LIN {X 0,Y 374.642,Z 535.942,A -85,B 0,C 180,E1 -12888.125,E2 -12888.125} C_VEL
LIN {X 0,Y 374.323,Z 532.294,A -85,B 0,C 180,E1 -12888.371,E2 -12888.371} C_VEL
LIN {X 0,Y 371.906,Z 526.656,A -85,B 0,C 180,E1 -12888.815,E2 -12888.815} C_VEL
LIN {X 0,Y 369.429,Z 520.933,A -85,B 0,C 180,E1 -12889.223,E2 -12889.223} C_VEL
LIN {X 0,Y 368.959,Z 517.153,A -85,B 0,C 180,E1 -12889.399,E2 -12889.399} C_VEL
LIN {X 0,Y 369.367,Z 505.054,A -85,B 0,C 180,E1 -12889.739,E2 -12889.739} C_VEL
LIN {X 0,Y 370.451,Z 429.303,A -85,B 0,C 180,E1 -12891.218,E2 -12891.218} C_VEL
LIN {X 0,Y 365.654,Z 406.161,A -85,B 0,C 180,E1 -12891.992,E2 -12891.992} C_VEL
LIN {X 0,Y 364.747,Z 403.294,A -85,B 0,C 180,E1 -12892.123,E2 -12892.123} C_VEL
LIN {X 0,Y 362.511,Z 391.552,A -85,B 0,C 180,E1 -12895.554,E2 -12895.554} C_VEL
LIN {X 0,Y 361.948,Z 388.902,A -85,B 0,C 180,E1 -12896.37,E2 -12896.37} C_VEL
LIN {X 0,Y 361.916,Z 388.903,A -85,B 0,C 180,E1 -12899.09,E2 -12899.09} C_VEL
LIN {X 0,Y 361.852,Z 388.912,A -85,B 0,C 180,E1 -12902.945,E2 -12902.945} C_VEL
LIN {X 0,Y 361.871,Z 388.905,A -85,B 0,C 180,E1 -12905.637,E2 -12905.637} C_VEL
LIN {X 0,Y 361.873,Z 388.908,A -85,B 0,C 180,E1 -12909.027,E2 -12909.027} C_VEL
LIN {X 0,Y 361.839,Z 388.913,A -85,B 0,C 180,E1 -12912.829,E2 -12912.829} C_VEL
LIN {X 0,Y 361.825,Z 388.912,A -85,B 0,C 180,E1 -12915.946,E2 -12915.946} C_VEL
LIN {X 0,Y 361.859,Z 388.907,A -85,B 0,C 180,E1 -12919.241,E2 -12919.241} C_VEL
LIN {X 0,Y 361.875,Z 388.908,A -85,B 0,C 180,E1 -12922.776,E2 -12922.776} C_VEL
LIN {X 0,Y 361.858,Z 388.907,A -85,B 0,C 180,E1 -12925.72,E2 -12925.72} C_VEL
LIN {X 0,Y 361.88,Z 388.905,A -85,B 0,C 180,E1 -12929.672,E2 -12929.672} C_VEL
LIN {X 0,Y 361.959,Z 388.895,A -85,B 0,C 180,E1 -12933.475,E2 -12933.475} C_VEL
LIN {X 0,Y 361.897,Z 388.902,A -85,B 0,C 180,E1 -12937.145,E2 -12937.145} C_VEL
LIN {X 0,Y 361.933,Z 388.898,A -85,B 0,C 180,E1 -12940.725,E2 -12940.725} C_VEL
LIN {X 0,Y 361.951,Z 388.9,A -85,B 0,C 180,E1 -12944.226,E2 -12944.226} C_VEL
LIN {X 0,Y 362.003,Z 388.89,A -85,B 0,C 180,E1 -12946.528,E2 -12946.528} C_VEL
LIN {X 0,Y 362.036,Z 388.891,A -85,B 0,C 180,E1 -12949.938,E2 -12949.938} C_VEL
LIN {X 0,Y 362.156,Z 388.873,A -85,B 0,C 180,E1 -12952.193,E2 -12952.193} C_VEL
LIN {X 0,Y 362.123,Z 388.875,A -85,B 0,C 180,E1 -12954.431,E2 -12954.431} C_VEL
LIN {X 0,Y 362.286,Z 388.859,A -85,B 0,C 180,E1 -12957.776,E2 -12957.776} C_VEL
LIN {X 0,Y 362.431,Z 388.84,A -85,B 0,C 180,E1 -12960,E2 -12960} C_VEL
LIN {X 0,Y 362.286,Z 388.856,A -85,B 0,C 180,E1 -12962.223,E2 -12962.223} C_VEL
LIN {X 0,Y 362.157,Z 388.87,A -85,B 0,C 180,E1 -12966.686,E2 -12966.686} C_VEL
LIN {X 0,Y 362.037,Z 388.887,A -85,B 0,C 180,E1 -12970.062,E2 -12970.062} C_VEL
LIN {X 0,Y 362.003,Z 388.892,A -85,B 0,C 180,E1 -12973.899,E2 -12973.899} C_VEL
LIN {X 0,Y 361.971,Z 388.895,A -85,B 0,C 180,E1 -12977.938,E2 -12977.938} C_VEL
LIN {X 0,Y 361.897,Z 388.906,A -85,B 0,C 180,E1 -12981.653,E2 -12981.653} C_VEL
LIN {X 0,Y 361.932,Z 388.903,A -85,B 0,C 180,E1 -12985.29,E2 -12985.29} C_VEL
LIN {X 0,Y 361.912,Z 388.902,A -85,B 0,C 180,E1 -12987.779,E2 -12987.779} C_VEL
LIN {X 0,Y 361.841,Z 388.912,A -85,B 0,C 180,E1 -12991.629,E2 -12991.629} C_VEL
LIN {X 0,Y 361.877,Z 388.91,A -85,B 0,C 180,E1 -12995.345,E2 -12995.345} C_VEL
LIN {X 0,Y 361.872,Z 388.91,A -85,B 0,C 180,E1 -12999.026,E2 -12999.026} C_VEL
LIN {X 0,Y 361.84,Z 388.912,A -85,B 0,C 180,E1 -13002.828,E2 -13002.828} C_VEL
LIN {X 0,Y 361.831,Z 388.91,A -85,B 0,C 180,E1 -13005.945,E2 -13005.945} C_VEL
LIN {X 0,Y 361.839,Z 388.913,A -85,B 0,C 180,E1 -13009.244,E2 -13009.244} C_VEL
LIN {X 0,Y 361.867,Z 388.91,A -85,B 0,C 180,E1 -13012.777,E2 -13012.777} C_VEL
LIN {X 0,Y 361.857,Z 388.907,A -85,B 0,C 180,E1 -13015.719,E2 -13015.719} C_VEL
LIN {X 0,Y 361.882,Z 388.909,A -85,B 0,C 180,E1 -13019.672,E2 -13019.672} C_VEL
LIN {X 0,Y 361.935,Z 389.076,A -85,B 0,C 180,E1 -13020.317,E2 -13020.317} C_VEL
LIN {X 0,Y 364.172,Z 399.647,A -85,B 0,C 180,E1 -13023.187,E2 -13023.187} C_VEL
LIN {X 0,Y 365.709,Z 407.696,A -85,B 0,C 180,E1 -13025.293,E2 -13025.293} C_VEL
LIN {X 0,Y 364.82,Z 417.446,A -85,B 0,C 180,E1 -13027.621,E2 -13027.621} C_VEL
LIN {X 0,Y 364.736,Z 418.695,A -85,B 0,C 180,E1 -13027.921,E2 -13027.921} C_VEL
LIN {X 0,Y 369.876,Z 448.618,A -85,B 0,C 180,E1 -13028.855,E2 -13028.855} C_VEL
LIN {X 0,Y 370.27,Z 453.848,A -85,B 0,C 180,E1 -13028.985,E2 -13028.985} C_VEL
LIN {X 0,Y 369.021,Z 526.846,A -85,B 0,C 180,E1 -13030.423,E2 -13030.423} C_VEL
LIN {X 0,Y 368.4,Z 539.299,A -85,B 0,C 180,E1 -13030.859,E2 -13030.859} C_VEL
LIN {X 0,Y 367.479,Z 552.192,A -85,B 0,C 180,E1 -13031.533,E2 -13031.533} C_VEL
LIN {X 0,Y 366.459,Z 564.435,A -85,B 0,C 180,E1 -13032.419,E2 -13032.419} C_VEL
LIN {X 0,Y 365.313,Z 576.016,A -85,B 0,C 180,E1 -13033.515,E2 -13033.515} C_VEL
LIN {X 0,Y 364.277,Z 586.157,A -85,B 0,C 180,E1 -13034.721,E2 -13034.721} C_VEL
LIN {X 0,Y 363.413,Z 594.976,A -85,B 0,C 180,E1 -13036.011,E2 -13036.011} C_VEL
LIN {X 0,Y 362.534,Z 602.845,A -85,B 0,C 180,E1 -13037.403,E2 -13037.403} C_VEL
LIN {X 0,Y 361.629,Z 610.529,A -85,B 0,C 180,E1 -13039.077,E2 -13039.077} C_VEL
LIN {X 0,Y 360.954,Z 617.618,A -85,B 0,C 180,E1 -13041.039,E2 -13041.039} C_VEL
LIN {X 0,Y 360.601,Z 622.335,A -85,B 0,C 180,E1 -13042.722,E2 -13042.722} C_VEL
LIN {X 0,Y 360.383,Z 625.939,A -85,B 0,C 180,E1 -13044.404,E2 -13044.404} C_VEL
LIN {X 0,Y 360.346,Z 627.799,A -85,B 0,C 180,E1 -13045.525,E2 -13045.525} C_VEL
LIN {X 0,Y 360.29,Z 629.193,A -85,B 0,C 180,E1 -13046.645,E2 -13046.645} C_VEL
LIN {X 0,Y 360.289,Z 630.795,A -85,B 0,C 180,E1 -13048.882,E2 -13048.882} C_VEL
LIN {X 0,Y 360.311,Z 631.01,A -85,B 0,C 180,E1 -13050,E2 -13050} C_VEL
LIN {X 0,Y 360.289,Z 630.792,A -85,B 0,C 180,E1 -13051.118,E2 -13051.118} C_VEL
LIN {X 0,Y 360.29,Z 629.185,A -85,B 0,C 180,E1 -13053.355,E2 -13053.355} C_VEL
LIN {X 0,Y 360.346,Z 627.787,A -85,B 0,C 180,E1 -13054.474,E2 -13054.474} C_VEL
LIN {X 0,Y 360.382,Z 625.21,A -85,B 0,C 180,E1 -13055.968,E2 -13055.968} C_VEL
LIN {X 0,Y 360.697,Z 620.874,A -85,B 0,C 180,E1 -13057.839,E2 -13057.839} C_VEL
LIN {X 0,Y 361.197,Z 614.761,A -85,B 0,C 180,E1 -13059.802,E2 -13059.802} C_VEL
LIN {X 0,Y 361.868,Z 608.085,A -85,B 0,C 180,E1 -13061.482,E2 -13061.482} C_VEL
LIN {X 0,Y 362.864,Z 599.806,A -85,B 0,C 180,E1 -13063.154,E2 -13063.154} C_VEL
LIN {X 0,Y 363.732,Z 591.315,A -85,B 0,C 180,E1 -13064.548,E2 -13064.548} C_VEL
LIN {X 0,Y 364.806,Z 580.824,A -85,B 0,C 180,E1 -13065.934,E2 -13065.934} C_VEL
LIN {X 0,Y 365.981,Z 569.017,A -85,B 0,C 180,E1 -13067.172,E2 -13067.172} C_VEL
LIN {X 0,Y 367.024,Z 557.134,A -85,B 0,C 180,E1 -13068.129,E2 -13068.129} C_VEL
LIN {X 0,Y 368.02,Z 544.771,A -85,B 0,C 180,E1 -13068.872,E2 -13068.872} C_VEL
LIN {X 0,Y 368.758,Z 532.06,A -85,B 0,C 180,E1 -13069.41,E2 -13069.41} C_VEL
LIN {X 0,Y 369.217,Z 518.696,A -85,B 0,C 180,E1 -13069.747,E2 -13069.747} C_VEL
LIN {X 0,Y 370.129,Z 450.447,A -85,B 0,C 180,E1 -13071.079,E2 -13071.079} C_VEL
LIN {X 0,Y 365.387,Z 422.391,A -85,B 0,C 180,E1 -13071.944,E2 -13071.944} C_VEL
LIN {X 0,Y 364.722,Z 418.661,A -85,B 0,C 180,E1 -13072.071,E2 -13072.071} C_VEL
LIN {X 0,Y 365.716,Z 408.872,A -85,B 0,C 180,E1 -13074.404,E2 -13074.404} C_VEL
LIN {X 0,Y 364.791,Z 402.605,A -85,B 0,C 180,E1 -13076.014,E2 -13076.014} C_VEL
LIN {X 0,Y 362.303,Z 390.756,A -85,B 0,C 180,E1 -13079.2,E2 -13079.2} C_VEL
LIN {X 0,Y 361.893,Z 388.903,A -85,B 0,C 180,E1 -13079.764,E2 -13079.764} C_VEL
LIN {X 0,Y 361.86,Z 388.91,A -85,B 0,C 180,E1 -13083.369,E2 -13083.369} C_VEL
LIN {X 0,Y 361.869,Z 388.912,A -85,B 0,C 180,E1 -13087.018,E2 -13087.018} C_VEL
LIN {X 0,Y 361.857,Z 388.907,A -85,B 0,C 180,E1 -13089.861,E2 -13089.861} C_VEL
LIN {X 0,Y 361.837,Z 388.915,A -85,B 0,C 180,E1 -13092.829,E2 -13092.829} C_VEL
LIN {X 0,Y 361.83,Z 388.91,A -85,B 0,C 180,E1 -13095.945,E2 -13095.945} C_VEL
LIN {X 0,Y 361.838,Z 388.912,A -85,B 0,C 180,E1 -13099.244,E2 -13099.244} C_VEL
LIN {X 0,Y 361.865,Z 388.912,A -85,B 0,C 180,E1 -13102.777,E2 -13102.777} C_VEL
LIN {X 0,Y 361.856,Z 388.907,A -85,B 0,C 180,E1 -13105.72,E2 -13105.72} C_VEL
LIN {X 0,Y 361.874,Z 388.905,A -85,B 0,C 180,E1 -13109.672,E2 -13109.672} C_VEL
LIN {X 0,Y 361.955,Z 388.895,A -85,B 0,C 180,E1 -13113.475,E2 -13113.475} C_VEL
LIN {X 0,Y 361.894,Z 388.904,A -85,B 0,C 180,E1 -13117.145,E2 -13117.145} C_VEL
LIN {X 0,Y 361.909,Z 388.905,A -85,B 0,C 180,E1 -13120.723,E2 -13120.723} C_VEL
LIN {X 0,Y 361.935,Z 388.898,A -85,B 0,C 180,E1 -13123.066,E2 -13123.066} C_VEL
LIN {X 0,Y 362.003,Z 388.894,A -85,B 0,C 180,E1 -13126.528,E2 -13126.528} C_VEL
LIN {X 0,Y 362.035,Z 388.887,A -85,B 0,C 180,E1 -13129.938,E2 -13129.938} C_VEL
LIN {X 0,Y 362.153,Z 388.87,A -85,B 0,C 180,E1 -13133.314,E2 -13133.314} C_VEL
LIN {X 0,Y 362.283,Z 388.856,A -85,B 0,C 180,E1 -13137.777,E2 -13137.777} C_VEL
LIN {X 0,Y 362.429,Z 388.84,A -85,B 0,C 180,E1 -13140,E2 -13140} C_VEL
LIN {X 0,Y 362.286,Z 388.86,A -85,B 0,C 180,E1 -13142.224,E2 -13142.224} C_VEL
LIN {X 0,Y 362.175,Z 388.868,A -85,B 0,C 180,E1 -13146.686,E2 -13146.686} C_VEL
LIN {X 0,Y 362.076,Z 388.88,A -85,B 0,C 180,E1 -13148.933,E2 -13148.933} C_VEL
LIN {X 0,Y 361.963,Z 388.897,A -85,B 0,C 180,E1 -13152.332,E2 -13152.332} C_VEL
LIN {X 0,Y 361.964,Z 388.894,A -85,B 0,C 180,E1 -13154.62,E2 -13154.62} C_VEL
LIN {X 0,Y 361.963,Z 388.898,A -85,B 0,C 180,E1 -13158.099,E2 -13158.099} C_VEL
LIN {X 0,Y 361.901,Z 388.905,A -85,B 0,C 180,E1 -13161.652,E2 -13161.652} C_VEL
LIN {X 0,Y 361.93,Z 388.899,A -85,B 0,C 180,E1 -13165.29,E2 -13165.29} C_VEL
LIN {X 0,Y 361.925,Z 388.905,A -85,B 0,C 180,E1 -13167.778,E2 -13167.778} C_VEL
LIN {X 0,Y 361.849,Z 388.91,A -85,B 0,C 180,E1 -13171.285,E2 -13171.285} C_VEL
LIN {X 0,Y 361.857,Z 388.908,A -85,B 0,C 180,E1 -13174.28,E2 -13174.28} C_VEL
LIN {X 0,Y 361.873,Z 388.907,A -85,B 0,C 180,E1 -13177.225,E2 -13177.225} C_VEL
LIN {X 0,Y 361.857,Z 388.907,A -85,B 0,C 180,E1 -13180.759,E2 -13180.759} C_VEL
LIN {X 0,Y 361.82,Z 388.912,A -85,B 0,C 180,E1 -13184.368,E2 -13184.368} C_VEL
LIN {X 0,Y 361.838,Z 388.915,A -85,B 0,C 180,E1 -13187.568,E2 -13187.568} C_VEL
LIN {X 0,Y 361.872,Z 388.907,A -85,B 0,C 180,E1 -13190.973,E2 -13190.973} C_VEL
LIN {X 0,Y 361.877,Z 388.905,A -85,B 0,C 180,E1 -13194.655,E2 -13194.655} C_VEL
LIN {X 0,Y 361.839,Z 388.909,A -85,B 0,C 180,E1 -13198.371,E2 -13198.371} C_VEL
LIN {X 0,Y 361.902,Z 388.905,A -85,B 0,C 180,E1 -13200.955,E2 -13200.955} C_VEL
LIN {X 0,Y 361.983,Z 389.022,A -85,B 0,C 180,E1 -13203.788,E2 -13203.788} C_VEL
LIN {X 0,Y 364.099,Z 399.857,A -85,B 0,C 180,E1 -13206.991,E2 -13206.991} C_VEL
LIN {X 0,Y 364.792,Z 403.485,A -85,B 0,C 180,E1 -13208.002,E2 -13208.002} C_VEL
LIN {X 0,Y 367.169,Z 412.809,A -85,B 0,C 180,E1 -13208.346,E2 -13208.346} C_VEL
LIN {X 0,Y 370.497,Z 429.487,A -85,B 0,C 180,E1 -13208.892,E2 -13208.892} C_VEL
LIN {X 0,Y 369.404,Z 500.103,A -85,B 0,C 180,E1 -13210.263,E2 -13210.263} C_VEL
LIN {X 0,Y 369.09,Z 514.346,A -85,B 0,C 180,E1 -13210.608,E2 -13210.608} C_VEL
LIN {X 0,Y 368.429,Z 526.232,A -85,B 0,C 180,E1 -13211.078,E2 -13211.078} C_VEL
LIN {X 0,Y 367.691,Z 538.092,A -85,B 0,C 180,E1 -13211.761,E2 -13211.761} C_VEL
LIN {X 0,Y 366.838,Z 548.926,A -85,B 0,C 180,E1 -13212.582,E2 -13212.582} C_VEL
LIN {X 0,Y 365.872,Z 559.858,A -85,B 0,C 180,E1 -13213.637,E2 -13213.637} C_VEL
LIN {X 0,Y 364.905,Z 570.515,A -85,B 0,C 180,E1 -13214.93,E2 -13214.93} C_VEL
LIN {X 0,Y 363.831,Z 579.7,A -85,B 0,C 180,E1 -13216.312,E2 -13216.312} C_VEL
LIN {X 0,Y 362.783,Z 588.618,A -85,B 0,C 180,E1 -13217.98,E2 -13217.98} C_VEL
LIN {X 0,Y 361.952,Z 595.798,A -85,B 0,C 180,E1 -13219.653,E2 -13219.653} C_VEL
LIN {X 0,Y 361.388,Z 600.639,A -85,B 0,C 180,E1 -13221.05,E2 -13221.05} C_VEL
LIN {X 0,Y 360.926,Z 605.343,A -85,B 0,C 180,E1 -13222.729,E2 -13222.729} C_VEL
LIN {X 0,Y 360.703,Z 608.941,A -85,B 0,C 180,E1 -13224.41,E2 -13224.41} C_VEL
LIN {X 0,Y 360.533,Z 610.802,A -85,B 0,C 180,E1 -13225.528,E2 -13225.528} C_VEL
LIN {X 0,Y 360.392,Z 612.203,A -85,B 0,C 180,E1 -13226.646,E2 -13226.646} C_VEL
LIN {X 0,Y 360.332,Z 613.811,A -85,B 0,C 180,E1 -13228.883,E2 -13228.883} C_VEL
LIN {X 0,Y 360.314,Z 614.043,A -85,B 0,C 180,E1 -13230,E2 -13230} C_VEL
LIN {X 0,Y 360.332,Z 613.853,A -85,B 0,C 180,E1 -13231.118,E2 -13231.118} C_VEL
LIN {X 0,Y 360.39,Z 612.301,A -85,B 0,C 180,E1 -13233.354,E2 -13233.354} C_VEL
LIN {X 0,Y 360.527,Z 610.942,A -85,B 0,C 180,E1 -13234.472,E2 -13234.472} C_VEL
LIN {X 0,Y 360.811,Z 607.155,A -85,B 0,C 180,E1 -13236.586,E2 -13236.586} C_VEL
LIN {X 0,Y 361.216,Z 602.625,A -85,B 0,C 180,E1 -13238.391,E2 -13238.391} C_VEL
LIN {X 0,Y 361.924,Z 596.182,A -85,B 0,C 180,E1 -13240.348,E2 -13240.348} C_VEL
LIN {X 0,Y 362.705,Z 589.103,A -85,B 0,C 180,E1 -13242.023,E2 -13242.023} C_VEL
LIN {X 0,Y 363.783,Z 580.28,A -85,B 0,C 180,E1 -13243.69,E2 -13243.69} C_VEL
LIN {X 0,Y 364.821,Z 571.225,A -85,B 0,C 180,E1 -13245.074,E2 -13245.074} C_VEL
LIN {X 0,Y 365.711,Z 561.582,A -85,B 0,C 180,E1 -13246.28,E2 -13246.28} C_VEL
LIN {X 0,Y 366.628,Z 551.626,A -85,B 0,C 180,E1 -13247.285,E2 -13247.285} C_VEL
LIN {X 0,Y 367.642,Z 539.509,A -85,B 0,C 180,E1 -13248.242,E2 -13248.242} C_VEL
LIN {X 0,Y 368.492,Z 526.812,A -85,B 0,C 180,E1 -13248.991,E2 -13248.991} C_VEL
LIN {X 0,Y 368.959,Z 517.153,A -85,B 0,C 180,E1 -13249.399,E2 -13249.399} C_VEL
LIN {X 0,Y 368.658,Z 511.429,A -85,B 0,C 180,E1 -13249.617,E2 -13249.617} C_VEL
LIN {X 0,Y 363.733,Z 492.736,A -85,B 0,C 180,E1 -13250.323,E2 -13250.323} C_VEL
LIN {X 0,Y 363.063,Z 486.919,A -85,B 0,C 180,E1 -13250.477,E2 -13250.477} C_VEL
LIN {X 0,Y 363.866,Z 430.386,A -85,B 0,C 180,E1 -13251.601,E2 -13251.601} C_VEL
LIN {X 0,Y 359.358,Z 408.508,A -85,B 0,C 180,E1 -13252.351,E2 -13252.351} C_VEL
LIN {X 0,Y 357.544,Z 403.4,A -85,B 0,C 180,E1 -13252.613,E2 -13252.613} C_VEL
LIN {X 0,Y 355.548,Z 392.794,A -85,B 0,C 180,E1 -13255.777,E2 -13255.777} C_VEL
LIN {X 0,Y 354.901,Z 389.782,A -85,B 0,C 180,E1 -13256.72,E2 -13256.72} C_VEL
LIN {X 0,Y 354.857,Z 389.78,A -85,B 0,C 180,E1 -13259.679,E2 -13259.679} C_VEL
LIN {X 0,Y 354.809,Z 389.785,A -85,B 0,C 180,E1 -13263.702,E2 -13263.702} C_VEL
LIN {X 0,Y 354.801,Z 389.79,A -85,B 0,C 180,E1 -13266.46,E2 -13266.46} C_VEL
LIN {X 0,Y 354.827,Z 389.783,A -85,B 0,C 180,E1 -13269.424,E2 -13269.424} C_VEL
LIN {X 0,Y 354.792,Z 389.791,A -85,B 0,C 180,E1 -13272.867,E2 -13272.867} C_VEL
LIN {X 0,Y 354.774,Z 389.791,A -85,B 0,C 180,E1 -13276.104,E2 -13276.104} C_VEL
LIN {X 0,Y 354.81,Z 389.785,A -85,B 0,C 180,E1 -13279.182,E2 -13279.182} C_VEL
LIN {X 0,Y 354.816,Z 389.789,A -85,B 0,C 180,E1 -13282.402,E2 -13282.402} C_VEL
LIN {X 0,Y 354.816,Z 389.785,A -85,B 0,C 180,E1 -13284.941,E2 -13284.941} C_VEL
LIN {X 0,Y 354.798,Z 389.792,A -85,B 0,C 180,E1 -13288.405,E2 -13288.405} C_VEL
LIN {X 0,Y 354.858,Z 389.779,A -85,B 0,C 180,E1 -13291.619,E2 -13291.619} C_VEL
LIN {X 0,Y 354.904,Z 389.779,A -85,B 0,C 180,E1 -13294.173,E2 -13294.173} C_VEL
LIN {X 0,Y 354.844,Z 389.784,A -85,B 0,C 180,E1 -13297.894,E2 -13297.894} C_VEL
LIN {X 0,Y 354.928,Z 389.773,A -85,B 0,C 180,E1 -13301.891,E2 -13301.891} C_VEL
LIN {X 0,Y 354.947,Z 389.773,A -85,B 0,C 180,E1 -13305.981,E2 -13305.981} C_VEL
LIN {X 0,Y 354.983,Z 389.767,A -85,B 0,C 180,E1 -13309.736,E2 -13309.736} C_VEL
LIN {X 0,Y 355.119,Z 389.751,A -85,B 0,C 180,E1 -13312.037,E2 -13312.037} C_VEL
LIN {X 0,Y 355.098,Z 389.751,A -85,B 0,C 180,E1 -13314.321,E2 -13314.321} C_VEL
LIN {X 0,Y 355.249,Z 389.735,A -85,B 0,C 180,E1 -13317.732,E2 -13317.732} C_VEL
LIN {X 0,Y 355.401,Z 389.716,A -85,B 0,C 180,E1 -13320,E2 -13320} C_VEL
LIN {X 0,Y 355.249,Z 389.732,A -85,B 0,C 180,E1 -13322.268,E2 -13322.268} C_VEL
LIN {X 0,Y 355.119,Z 389.746,A -85,B 0,C 180,E1 -13326.82,E2 -13326.82} C_VEL
LIN {X 0,Y 354.985,Z 389.764,A -85,B 0,C 180,E1 -13330.264,E2 -13330.264} C_VEL
LIN {X 0,Y 354.948,Z 389.77,A -85,B 0,C 180,E1 -13334.019,E2 -13334.019} C_VEL
LIN {X 0,Y 354.926,Z 389.771,A -85,B 0,C 180,E1 -13338.108,E2 -13338.108} C_VEL
LIN {X 0,Y 354.84,Z 389.781,A -85,B 0,C 180,E1 -13342.106,E2 -13342.106} C_VEL
LIN {X 0,Y 354.903,Z 389.776,A -85,B 0,C 180,E1 -13345.827,E2 -13345.827} C_VEL
LIN {X 0,Y 354.821,Z 389.786,A -85,B 0,C 180,E1 -13349.682,E2 -13349.682} C_VEL
LIN {X 0,Y 354.809,Z 389.787,A -85,B 0,C 180,E1 -13353.702,E2 -13353.702} C_VEL
LIN {X 0,Y 354.801,Z 389.786,A -85,B 0,C 180,E1 -13356.459,E2 -13356.459} C_VEL
LIN {X 0,Y 354.827,Z 389.787,A -85,B 0,C 180,E1 -13359.423,E2 -13359.423} C_VEL
LIN {X 0,Y 354.792,Z 389.791,A -85,B 0,C 180,E1 -13362.867,E2 -13362.867} C_VEL
LIN {X 0,Y 354.778,Z 389.789,A -85,B 0,C 180,E1 -13366.105,E2 -13366.105} C_VEL
LIN {X 0,Y 354.791,Z 389.792,A -85,B 0,C 180,E1 -13369.179,E2 -13369.179} C_VEL
LIN {X 0,Y 354.81,Z 389.786,A -85,B 0,C 180,E1 -13372.402,E2 -13372.402} C_VEL
LIN {X 0,Y 354.815,Z 389.79,A -85,B 0,C 180,E1 -13374.941,E2 -13374.941} C_VEL
LIN {X 0,Y 354.796,Z 389.789,A -85,B 0,C 180,E1 -13378.405,E2 -13378.405} C_VEL
LIN {X 0,Y 354.861,Z 389.854,A -85,B 0,C 180,E1 -13379.913,E2 -13379.913} C_VEL
LIN {X 0,Y 356.956,Z 399.523,A -85,B 0,C 180,E1 -13382.609,E2 -13382.609} C_VEL
LIN {X 0,Y 358.731,Z 408.764,A -85,B 0,C 180,E1 -13385.088,E2 -13385.088} C_VEL
LIN {X 0,Y 358.322,Z 414.903,A -85,B 0,C 180,E1 -13386.598,E2 -13386.598} C_VEL
LIN {X 0,Y 357.88,Z 418.453,A -85,B 0,C 180,E1 -13387.457,E2 -13387.457} C_VEL
LIN {X 0,Y 362.199,Z 442.899,A -85,B 0,C 180,E1 -13388.269,E2 -13388.269} C_VEL
LIN {X 0,Y 363.652,Z 453.269,A -85,B 0,C 180,E1 -13388.575,E2 -13388.575} C_VEL
LIN {X 0,Y 362.349,Z 526.692,A -85,B 0,C 180,E1 -13390.047,E2 -13390.047} C_VEL
LIN {X 0,Y 361.715,Z 539.141,A -85,B 0,C 180,E1 -13390.491,E2 -13390.491} C_VEL
LIN {X 0,Y 360.76,Z 552.031,A -85,B 0,C 180,E1 -13391.176,E2 -13391.176} C_VEL
LIN {X 0,Y 359.699,Z 564.272,A -85,B 0,C 180,E1 -13392.077,E2 -13392.077} C_VEL
LIN {X 0,Y 358.508,Z 575.853,A -85,B 0,C 180,E1 -13393.193,E2 -13393.193} C_VEL
LIN {X 0,Y 357.522,Z 584.907,A -85,B 0,C 180,E1 -13394.277,E2 -13394.277} C_VEL
LIN {X 0,Y 356.485,Z 594.811,A -85,B 0,C 180,E1 -13395.733,E2 -13395.733} C_VEL
LIN {X 0,Y 355.588,Z 602.679,A -85,B 0,C 180,E1 -13397.153,E2 -13397.153} C_VEL
LIN {X 0,Y 354.62,Z 610.362,A -85,B 0,C 180,E1 -13398.858,E2 -13398.858} C_VEL
LIN {X 0,Y 353.906,Z 617.451,A -85,B 0,C 180,E1 -13400.859,E2 -13400.859} C_VEL
LIN {X 0,Y 353.525,Z 622.168,A -85,B 0,C 180,E1 -13402.575,E2 -13402.575} C_VEL
LIN {X 0,Y 353.282,Z 625.772,A -85,B 0,C 180,E1 -13404.291,E2 -13404.291} C_VEL
LIN {X 0,Y 353.261,Z 627.632,A -85,B 0,C 180,E1 -13405.435,E2 -13405.435} C_VEL
LIN {X 0,Y 353.212,Z 629.026,A -85,B 0,C 180,E1 -13406.578,E2 -13406.578} C_VEL
LIN {X 0,Y 353.189,Z 630.628,A -85,B 0,C 180,E1 -13408.86,E2 -13408.86} C_VEL
LIN {X 0,Y 353.213,Z 630.843,A -85,B 0,C 180,E1 -13410,E2 -13410} C_VEL
LIN {X 0,Y 353.189,Z 630.624,A -85,B 0,C 180,E1 -13411.14,E2 -13411.14} C_VEL
LIN {X 0,Y 353.212,Z 629.018,A -85,B 0,C 180,E1 -13413.422,E2 -13413.422} C_VEL
LIN {X 0,Y 353.261,Z 627.62,A -85,B 0,C 180,E1 -13414.564,E2 -13414.564} C_VEL
LIN {X 0,Y 353.296,Z 625.325,A -85,B 0,C 180,E1 -13415.937,E2 -13415.937} C_VEL
LIN {X 0,Y 353.637,Z 620.705,A -85,B 0,C 180,E1 -13417.996,E2 -13417.996} C_VEL
LIN {X 0,Y 354.178,Z 614.592,A -85,B 0,C 180,E1 -13419.999,E2 -13419.999} C_VEL
LIN {X 0,Y 354.892,Z 607.916,A -85,B 0,C 180,E1 -13421.711,E2 -13421.711} C_VEL
LIN {X 0,Y 355.936,Z 599.636,A -85,B 0,C 180,E1 -13423.415,E2 -13423.415} C_VEL
LIN {X 0,Y 356.963,Z 590.049,A -85,B 0,C 180,E1 -13424.994,E2 -13424.994} C_VEL
LIN {X 0,Y 358.071,Z 579.476,A -85,B 0,C 180,E1 -13426.388,E2 -13426.388} C_VEL
LIN {X 0,Y 359.201,Z 568.845,A -85,B 0,C 180,E1 -13427.507,E2 -13427.507} C_VEL
LIN {X 0,Y 360.276,Z 556.961,A -85,B 0,C 180,E1 -13428.481,E2 -13428.481} C_VEL
LIN {X 0,Y 361.308,Z 544.596,A -85,B 0,C 180,E1 -13429.236,E2 -13429.236} C_VEL
LIN {X 0,Y 362.075,Z 531.882,A -85,B 0,C 180,E1 -13429.783,E2 -13429.783} C_VEL
LIN {X 0,Y 362.552,Z 518.509,A -85,B 0,C 180,E1 -13430.126,E2 -13430.126} C_VEL
LIN {X 0,Y 363.463,Z 450.944,A -85,B 0,C 180,E1 -13431.47,E2 -13431.47} C_VEL
LIN {X 0,Y 358.713,Z 422.976,A -85,B 0,C 180,E1 -13432.357,E2 -13432.357} C_VEL
LIN {X 0,Y 357.893,Z 418.441,A -85,B 0,C 180,E1 -13432.527,E2 -13432.527} C_VEL
LIN {X 0,Y 358.792,Z 409.931,A -85,B 0,C 180,E1 -13434.598,E2 -13434.598} C_VEL
LIN {X 0,Y 357.548,Z 402.508,A -85,B 0,C 180,E1 -13436.563,E2 -13436.563} C_VEL
LIN {X 0,Y 355.18,Z 391.335,A -85,B 0,C 180,E1 -13439.648,E2 -13439.648} C_VEL
LIN {X 0,Y 354.842,Z 389.781,A -85,B 0,C 180,E1 -13440.13,E2 -13440.13} C_VEL
LIN {X 0,Y 354.807,Z 389.787,A -85,B 0,C 180,E1 -13443.702,E2 -13443.702} C_VEL
LIN {X 0,Y 354.799,Z 389.787,A -85,B 0,C 180,E1 -13446.459,E2 -13446.459} C_VEL
LIN {X 0,Y 354.825,Z 389.785,A -85,B 0,C 180,E1 -13449.424,E2 -13449.424} C_VEL
LIN {X 0,Y 354.79,Z 389.793,A -85,B 0,C 180,E1 -13452.867,E2 -13452.867} C_VEL
LIN {X 0,Y 354.777,Z 389.789,A -85,B 0,C 180,E1 -13456.105,E2 -13456.105} C_VEL
LIN {X 0,Y 354.79,Z 389.79,A -85,B 0,C 180,E1 -13459.179,E2 -13459.179} C_VEL
LIN {X 0,Y 354.809,Z 389.787,A -85,B 0,C 180,E1 -13462.402,E2 -13462.402} C_VEL
LIN {X 0,Y 354.813,Z 389.789,A -85,B 0,C 180,E1 -13464.941,E2 -13464.941} C_VEL
LIN {X 0,Y 354.795,Z 389.79,A -85,B 0,C 180,E1 -13468.405,E2 -13468.405} C_VEL
LIN {X 0,Y 354.848,Z 389.78,A -85,B 0,C 180,E1 -13471.619,E2 -13471.619} C_VEL
LIN {X 0,Y 354.901,Z 389.776,A -85,B 0,C 180,E1 -13474.173,E2 -13474.173} C_VEL
LIN {X 0,Y 354.838,Z 389.782,A -85,B 0,C 180,E1 -13477.894,E2 -13477.894} C_VEL
LIN {X 0,Y 354.924,Z 389.772,A -85,B 0,C 180,E1 -13481.892,E2 -13481.892} C_VEL
LIN {X 0,Y 354.945,Z 389.769,A -85,B 0,C 180,E1 -13485.981,E2 -13485.981} C_VEL
LIN {X 0,Y 354.983,Z 389.764,A -85,B 0,C 180,E1 -13489.736,E2 -13489.736} C_VEL
LIN {X 0,Y 355.116,Z 389.747,A -85,B 0,C 180,E1 -13493.18,E2 -13493.18} C_VEL
LIN {X 0,Y 355.246,Z 389.732,A -85,B 0,C 180,E1 -13497.732,E2 -13497.732} C_VEL
LIN {X 0,Y 355.398,Z 389.716,A -85,B 0,C 180,E1 -13500,E2 -13500} C_VEL
LIN {X 0,Y 355.249,Z 389.736,A -85,B 0,C 180,E1 -13502.268,E2 -13502.268} C_VEL
LIN {X 0,Y 355.141,Z 389.744,A -85,B 0,C 180,E1 -13506.819,E2 -13506.819} C_VEL
LIN {X 0,Y 355.017,Z 389.759,A -85,B 0,C 180,E1 -13509.112,E2 -13509.112} C_VEL
LIN {X 0,Y 354.923,Z 389.772,A -85,B 0,C 180,E1 -13512.581,E2 -13512.581} C_VEL
LIN {X 0,Y 354.892,Z 389.779,A -85,B 0,C 180,E1 -13516.096,E2 -13516.096} C_VEL
LIN {X 0,Y 354.911,Z 389.774,A -85,B 0,C 180,E1 -13518.472,E2 -13518.472} C_VEL
LIN {X 0,Y 354.841,Z 389.785,A -85,B 0,C 180,E1 -13522.106,E2 -13522.106} C_VEL
LIN {X 0,Y 354.902,Z 389.779,A -85,B 0,C 180,E1 -13525.827,E2 -13525.827} C_VEL
LIN {X 0,Y 354.856,Z 389.785,A -85,B 0,C 180,E1 -13529.679,E2 -13529.679} C_VEL
LIN {X 0,Y 354.808,Z 389.791,A -85,B 0,C 180,E1 -13533.702,E2 -13533.702} C_VEL
LIN {X 0,Y 354.803,Z 389.786,A -85,B 0,C 180,E1 -13536.459,E2 -13536.459} C_VEL
LIN {X 0,Y 354.825,Z 389.787,A -85,B 0,C 180,E1 -13539.424,E2 -13539.424} C_VEL
LIN {X 0,Y 354.792,Z 389.788,A -85,B 0,C 180,E1 -13542.868,E2 -13542.868} C_VEL
LIN {X 0,Y 354.769,Z 389.791,A -85,B 0,C 180,E1 -13546.104,E2 -13546.104} C_VEL
LIN {X 0,Y 354.79,Z 389.791,A -85,B 0,C 180,E1 -13549.179,E2 -13549.179} C_VEL
LIN {X 0,Y 354.81,Z 389.785,A -85,B 0,C 180,E1 -13552.402,E2 -13552.402} C_VEL
LIN {X 0,Y 354.815,Z 389.787,A -85,B 0,C 180,E1 -13554.941,E2 -13554.941} C_VEL
LIN {X 0,Y 354.795,Z 389.787,A -85,B 0,C 180,E1 -13558.405,E2 -13558.405} C_VEL
LIN {X 0,Y 354.853,Z 389.782,A -85,B 0,C 180,E1 -13561.619,E2 -13561.619} C_VEL
LIN {X 0,Y 354.929,Z 389.832,A -85,B 0,C 180,E1 -13563.413,E2 -13563.413} C_VEL
LIN {X 0,Y 357.141,Z 401.119,A -85,B 0,C 180,E1 -13566.823,E2 -13566.823} C_VEL
LIN {X 0,Y 357.61,Z 403.624,A -85,B 0,C 180,E1 -13567.535,E2 -13567.535} C_VEL
LIN {X 0,Y 360.081,Z 411.534,A -85,B 0,C 180,E1 -13567.866,E2 -13567.866} C_VEL
LIN {X 0,Y 363.939,Z 430.874,A -85,B 0,C 180,E1 -13568.518,E2 -13568.518} C_VEL
LIN {X 0,Y 362.678,Z 502.084,A -85,B 0,C 180,E1 -13569.919,E2 -13569.919} C_VEL
LIN {X 0,Y 362.375,Z 515.617,A -85,B 0,C 180,E1 -13570.271,E2 -13570.271} C_VEL
LIN {X 0,Y 361.685,Z 527.731,A -85,B 0,C 180,E1 -13570.785,E2 -13570.785} C_VEL
LIN {X 0,Y 360.825,Z 540.251,A -85,B 0,C 180,E1 -13571.548,E2 -13571.548} C_VEL
LIN {X 0,Y 359.82,Z 552.247,A -85,B 0,C 180,E1 -13572.524,E2 -13572.524} C_VEL
LIN {X 0,Y 358.835,Z 562.671,A -85,B 0,C 180,E1 -13573.616,E2 -13573.616} C_VEL
LIN {X 0,Y 357.825,Z 572.644,A -85,B 0,C 180,E1 -13574.916,E2 -13574.916} C_VEL
LIN {X 0,Y 356.725,Z 581.491,A -85,B 0,C 180,E1 -13576.325,E2 -13576.325} C_VEL
LIN {X 0,Y 355.689,Z 590.119,A -85,B 0,C 180,E1 -13578.026,E2 -13578.026} C_VEL
LIN {X 0,Y 354.853,Z 596.997,A -85,B 0,C 180,E1 -13579.732,E2 -13579.732} C_VEL
LIN {X 0,Y 354.197,Z 602.503,A -85,B 0,C 180,E1 -13581.442,E2 -13581.442} C_VEL
LIN {X 0,Y 353.72,Z 607.435,A -85,B 0,C 180,E1 -13583.437,E2 -13583.437} C_VEL
LIN {X 0,Y 353.473,Z 610.969,A -85,B 0,C 180,E1 -13585.439,E2 -13585.439} C_VEL
LIN {X 0,Y 353.314,Z 612.37,A -85,B 0,C 180,E1 -13586.579,E2 -13586.579} C_VEL
LIN {X 0,Y 353.234,Z 613.978,A -85,B 0,C 180,E1 -13588.86,E2 -13588.86} C_VEL
LIN {X 0,Y 353.217,Z 614.211,A -85,B 0,C 180,E1 -13590,E2 -13590} C_VEL
LIN {X 0,Y 353.234,Z 614.02,A -85,B 0,C 180,E1 -13591.14,E2 -13591.14} C_VEL
LIN {X 0,Y 353.312,Z 612.467,A -85,B 0,C 180,E1 -13593.421,E2 -13593.421} C_VEL
LIN {X 0,Y 353.467,Z 611.108,A -85,B 0,C 180,E1 -13594.562,E2 -13594.562} C_VEL
LIN {X 0,Y 353.719,Z 607.657,A -85,B 0,C 180,E1 -13596.562,E2 -13596.562} C_VEL
LIN {X 0,Y 354.192,Z 602.79,A -85,B 0,C 180,E1 -13598.559,E2 -13598.559} C_VEL
LIN {X 0,Y 354.908,Z 596.348,A -85,B 0,C 180,E1 -13600.555,E2 -13600.555} C_VEL
LIN {X 0,Y 355.747,Z 589.268,A -85,B 0,C 180,E1 -13602.262,E2 -13602.262} C_VEL
LIN {X 0,Y 356.886,Z 580.444,A -85,B 0,C 180,E1 -13603.96,E2 -13603.96} C_VEL
LIN {X 0,Y 357.967,Z 571.437,A -85,B 0,C 180,E1 -13605.363,E2 -13605.363} C_VEL
LIN {X 0,Y 358.996,Z 560.335,A -85,B 0,C 180,E1 -13606.755,E2 -13606.755} C_VEL
LIN {X 0,Y 360.144,Z 548.631,A -85,B 0,C 180,E1 -13607.9,E2 -13607.9} C_VEL
LIN {X 0,Y 361.182,Z 536.633,A -85,B 0,C 180,E1 -13608.801,E2 -13608.801} C_VEL
LIN {X 0,Y 361.971,Z 523.251,A -85,B 0,C 180,E1 -13609.531,E2 -13609.531} C_VEL
LIN {X 0,Y 362.579,Z 509.696,A -85,B 0,C 180,E1 -13610.014,E2 -13610.014} C_VEL
LIN {X 0,Y 363.063,Z 486.919,A -85,B 0,C 180,E1 -13610.477,E2 -13610.477} C_VEL
LIN {X 0,Y 362.416,Z 481.122,A -85,B 0,C 180,E1 -13610.636,E2 -13610.636} C_VEL
LIN {X 0,Y 357.466,Z 462.43,A -85,B 0,C 180,E1 -13611.332,E2 -13611.332} C_VEL
LIN {X 0,Y 356.95,Z 456.628,A -85,B 0,C 180,E1 -13611.487,E2 -13611.487} C_VEL
LIN {X 0,Y 357.298,Z 431.462,A -85,B 0,C 180,E1 -13611.999,E2 -13611.999} C_VEL
LIN {X 0,Y 353.082,Z 410.97,A -85,B 0,C 180,E1 -13612.72,E2 -13612.72} C_VEL
LIN {X 0,Y 350.41,Z 403.632,A -85,B 0,C 180,E1 -13613.083,E2 -13613.083} C_VEL
LIN {X 0,Y 348.586,Z 394.153,A -85,B 0,C 180,E1 -13615.977,E2 -13615.977} C_VEL
LIN {X 0,Y 347.845,Z 390.658,A -85,B 0,C 180,E1 -13617.135,E2 -13617.135} C_VEL
LIN {X 0,Y 347.767,Z 390.665,A -85,B 0,C 180,E1 -13620.347,E2 -13620.347} C_VEL
LIN {X 0,Y 347.748,Z 390.669,A -85,B 0,C 180,E1 -13624.464,E2 -13624.464} C_VEL
LIN {X 0,Y 347.777,Z 390.662,A -85,B 0,C 180,E1 -13627.989,E2 -13627.989} C_VEL
LIN {X 0,Y 347.754,Z 390.664,A -85,B 0,C 180,E1 -13631.83,E2 -13631.83} C_VEL
LIN {X 0,Y 347.769,Z 390.664,A -85,B 0,C 180,E1 -13635.017,E2 -13635.017} C_VEL
LIN {X 0,Y 347.761,Z 390.668,A -85,B 0,C 180,E1 -13638.396,E2 -13638.396} C_VEL
LIN {X 0,Y 347.781,Z 390.661,A -85,B 0,C 180,E1 -13642.011,E2 -13642.011} C_VEL
LIN {X 0,Y 347.748,Z 390.664,A -85,B 0,C 180,E1 -13645.536,E2 -13645.536} C_VEL
LIN {X 0,Y 347.768,Z 390.663,A -85,B 0,C 180,E1 -13649.654,E2 -13649.654} C_VEL
LIN {X 0,Y 347.857,Z 390.653,A -85,B 0,C 180,E1 -13652.744,E2 -13652.744} C_VEL
LIN {X 0,Y 347.794,Z 390.663,A -85,B 0,C 180,E1 -13656.162,E2 -13656.162} C_VEL
LIN {X 0,Y 347.832,Z 390.658,A -85,B 0,C 180,E1 -13659.91,E2 -13659.91} C_VEL
LIN {X 0,Y 347.872,Z 390.653,A -85,B 0,C 180,E1 -13662.359,E2 -13662.359} C_VEL
LIN {X 0,Y 347.902,Z 390.65,A -85,B 0,C 180,E1 -13665.971,E2 -13665.971} C_VEL
LIN {X 0,Y 347.933,Z 390.643,A -85,B 0,C 180,E1 -13669.526,E2 -13669.526} C_VEL
LIN {X 0,Y 348.079,Z 390.628,A -85,B 0,C 180,E1 -13671.875,E2 -13671.875} C_VEL
LIN {X 0,Y 348.073,Z 390.627,A -85,B 0,C 180,E1 -13674.206,E2 -13674.206} C_VEL
LIN {X 0,Y 348.211,Z 390.611,A -85,B 0,C 180,E1 -13677.686,E2 -13677.686} C_VEL
LIN {X 0,Y 348.35,Z 390.594,A -85,B 0,C 180,E1 -13680,E2 -13680} C_VEL
LIN {X 0,Y 348.211,Z 390.608,A -85,B 0,C 180,E1 -13682.313,E2 -13682.313} C_VEL
LIN {X 0,Y 348.087,Z 390.622,A -85,B 0,C 180,E1 -13686.958,E2 -13686.958} C_VEL
LIN {X 0,Y 347.936,Z 390.641,A -85,B 0,C 180,E1 -13690.474,E2 -13690.474} C_VEL
LIN {X 0,Y 347.903,Z 390.647,A -85,B 0,C 180,E1 -13694.15,E2 -13694.15} C_VEL
LIN {X 0,Y 347.895,Z 390.646,A -85,B 0,C 180,E1 -13698.29,E2 -13698.29} C_VEL
LIN {X 0,Y 347.794,Z 390.662,A -85,B 0,C 180,E1 -13701.636,E2 -13701.636} C_VEL
LIN {X 0,Y 347.817,Z 390.659,A -85,B 0,C 180,E1 -13705.108,E2 -13705.108} C_VEL
LIN {X 0,Y 347.812,Z 390.66,A -85,B 0,C 180,E1 -13707.694,E2 -13707.694} C_VEL
LIN {X 0,Y 347.753,Z 390.664,A -85,B 0,C 180,E1 -13710.348,E2 -13710.348} C_VEL
LIN {X 0,Y 347.751,Z 390.664,A -85,B 0,C 180,E1 -13714.044,E2 -13714.044} C_VEL
LIN {X 0,Y 347.765,Z 390.668,A -85,B 0,C 180,E1 -13717.321,E2 -13717.321} C_VEL
LIN {X 0,Y 347.736,Z 390.666,A -85,B 0,C 180,E1 -13720.297,E2 -13720.297} C_VEL
LIN {X 0,Y 347.729,Z 390.671,A -85,B 0,C 180,E1 -13723.407,E2 -13723.407} C_VEL
LIN {X 0,Y 347.73,Z 390.67,A -85,B 0,C 180,E1 -13726.686,E2 -13726.686} C_VEL
LIN {X 0,Y 347.75,Z 390.665,A -85,B 0,C 180,E1 -13730.173,E2 -13730.173} C_VEL
LIN {X 0,Y 347.765,Z 390.666,A -85,B 0,C 180,E1 -13732.679,E2 -13732.679} C_VEL
LIN {X 0,Y 347.751,Z 390.665,A -85,B 0,C 180,E1 -13735.956,E2 -13735.956} C_VEL
LIN {X 0,Y 347.804,Z 390.774,A -85,B 0,C 180,E1 -13739.531,E2 -13739.531} C_VEL
LIN {X 0,Y 350.094,Z 401.169,A -85,B 0,C 180,E1 -13742.502,E2 -13742.502} C_VEL
LIN {X 0,Y 351.885,Z 411.062,A -85,B 0,C 180,E1 -13745.202,E2 -13745.202} C_VEL
LIN {X 0,Y 351.091,Z 418.292,A -85,B 0,C 180,E1 -13746.997,E2 -13746.997} C_VEL
LIN {X 0,Y 355.636,Z 444.01,A -85,B 0,C 180,E1 -13747.874,E2 -13747.874} C_VEL
LIN {X 0,Y 357.052,Z 453.549,A -85,B 0,C 180,E1 -13748.168,E2 -13748.168} C_VEL
LIN {X 0,Y 355.664,Z 526.538,A -85,B 0,C 180,E1 -13749.656,E2 -13749.656} C_VEL
LIN {X 0,Y 354.981,Z 539.745,A -85,B 0,C 180,E1 -13750.143,E2 -13750.143} C_VEL
LIN {X 0,Y 353.95,Z 552.987,A -85,B 0,C 180,E1 -13750.875,E2 -13750.875} C_VEL
LIN {X 0,Y 352.928,Z 564.109,A -85,B 0,C 180,E1 -13751.721,E2 -13751.721} C_VEL
LIN {X 0,Y 351.708,Z 575.689,A -85,B 0,C 180,E1 -13752.858,E2 -13752.858} C_VEL
LIN {X 0,Y 350.606,Z 585.205,A -85,B 0,C 180,E1 -13754.023,E2 -13754.023} C_VEL
LIN {X 0,Y 349.558,Z 594.645,A -85,B 0,C 180,E1 -13755.444,E2 -13755.444} C_VEL
LIN {X 0,Y 348.63,Z 602.513,A -85,B 0,C 180,E1 -13756.892,E2 -13756.892} C_VEL
LIN {X 0,Y 347.602,Z 610.195,A -85,B 0,C 180,E1 -13758.631,E2 -13758.631} C_VEL
LIN {X 0,Y 346.876,Z 617.285,A -85,B 0,C 180,E1 -13760.672,E2 -13760.672} C_VEL
LIN {X 0,Y 346.475,Z 622.001,A -85,B 0,C 180,E1 -13762.423,E2 -13762.423} C_VEL
LIN {X 0,Y 346.201,Z 625.605,A -85,B 0,C 180,E1 -13764.174,E2 -13764.174} C_VEL
LIN {X 0,Y 346.158,Z 627.465,A -85,B 0,C 180,E1 -13765.342,E2 -13765.342} C_VEL
LIN {X 0,Y 346.136,Z 628.86,A -85,B 0,C 180,E1 -13766.508,E2 -13766.508} C_VEL
LIN {X 0,Y 346.089,Z 630.461,A -85,B 0,C 180,E1 -13768.836,E2 -13768.836} C_VEL
LIN {X 0,Y 346.115,Z 630.676,A -85,B 0,C 180,E1 -13770,E2 -13770} C_VEL
LIN {X 0,Y 346.089,Z 630.457,A -85,B 0,C 180,E1 -13771.163,E2 -13771.163} C_VEL
LIN {X 0,Y 346.136,Z 628.851,A -85,B 0,C 180,E1 -13773.492,E2 -13773.492} C_VEL
LIN {X 0,Y 346.159,Z 627.451,A -85,B 0,C 180,E1 -13774.658,E2 -13774.658} C_VEL
LIN {X 0,Y 346.26,Z 624.513,A -85,B 0,C 180,E1 -13776.409,E2 -13776.409} C_VEL
LIN {X 0,Y 346.578,Z 620.536,A -85,B 0,C 180,E1 -13778.16,E2 -13778.16} C_VEL
LIN {X 0,Y 347.149,Z 614.423,A -85,B 0,C 180,E1 -13780.203,E2 -13780.203} C_VEL
LIN {X 0,Y 347.913,Z 607.746,A -85,B 0,C 180,E1 -13781.95,E2 -13781.95} C_VEL
LIN {X 0,Y 349.01,Z 599.467,A -85,B 0,C 180,E1 -13783.686,E2 -13783.686} C_VEL
LIN {X 0,Y 349.964,Z 590.974,A -85,B 0,C 180,E1 -13785.133,E2 -13785.133} C_VEL
LIN {X 0,Y 351.108,Z 580.481,A -85,B 0,C 180,E1 -13786.573,E2 -13786.573} C_VEL
LIN {X 0,Y 352.416,Z 568.674,A -85,B 0,C 180,E1 -13787.855,E2 -13787.855} C_VEL
LIN {X 0,Y 353.565,Z 556.789,A -85,B 0,C 180,E1 -13788.845,E2 -13788.845} C_VEL
LIN {X 0,Y 354.61,Z 544.422,A -85,B 0,C 180,E1 -13789.614,E2 -13789.614} C_VEL
LIN {X 0,Y 355.408,Z 531.705,A -85,B 0,C 180,E1 -13790.171,E2 -13790.171} C_VEL
LIN {X 0,Y 355.908,Z 518.322,A -85,B 0,C 180,E1 -13790.518,E2 -13790.518} C_VEL
LIN {X 0,Y 356.886,Z 451.911,A -85,B 0,C 180,E1 -13791.862,E2 -13791.862} C_VEL
LIN {X 0,Y 352.163,Z 424.16,A -85,B 0,C 180,E1 -13792.767,E2 -13792.767} C_VEL
LIN {X 0,Y 351.094,Z 418.272,A -85,B 0,C 180,E1 -13792.989,E2 -13792.989} C_VEL
LIN {X 0,Y 351.859,Z 410.99,A -85,B 0,C 180,E1 -13794.8,E2 -13794.8} C_VEL
LIN {X 0,Y 350.08,Z 401.092,A -85,B 0,C 180,E1 -13797.499,E2 -13797.499} C_VEL
LIN {X 0,Y 347.795,Z 390.66,A -85,B 0,C 180,E1 -13800.511,E2 -13800.511} C_VEL
LIN {X 0,Y 347.746,Z 390.667,A -85,B 0,C 180,E1 -13804.464,E2 -13804.464} C_VEL
LIN {X 0,Y 347.775,Z 390.662,A -85,B 0,C 180,E1 -13807.989,E2 -13807.989} C_VEL
LIN {X 0,Y 347.752,Z 390.664,A -85,B 0,C 180,E1 -13811.83,E2 -13811.83} C_VEL
LIN {X 0,Y 347.767,Z 390.667,A -85,B 0,C 180,E1 -13815.017,E2 -13815.017} C_VEL
LIN {X 0,Y 347.752,Z 390.666,A -85,B 0,C 180,E1 -13818.397,E2 -13818.397} C_VEL
LIN {X 0,Y 347.775,Z 390.661,A -85,B 0,C 180,E1 -13822.011,E2 -13822.011} C_VEL
LIN {X 0,Y 347.745,Z 390.665,A -85,B 0,C 180,E1 -13825.536,E2 -13825.536} C_VEL
LIN {X 0,Y 347.746,Z 390.667,A -85,B 0,C 180,E1 -13828.3,E2 -13828.3} C_VEL
LIN {X 0,Y 347.78,Z 390.663,A -85,B 0,C 180,E1 -13830.988,E2 -13830.988} C_VEL
LIN {X 0,Y 347.832,Z 390.654,A -85,B 0,C 180,E1 -13833.608,E2 -13833.608} C_VEL
LIN {X 0,Y 347.791,Z 390.661,A -85,B 0,C 180,E1 -13836.162,E2 -13836.162} C_VEL
LIN {X 0,Y 347.815,Z 390.657,A -85,B 0,C 180,E1 -13839.909,E2 -13839.909} C_VEL
LIN {X 0,Y 347.868,Z 390.654,A -85,B 0,C 180,E1 -13842.359,E2 -13842.359} C_VEL
LIN {X 0,Y 347.899,Z 390.647,A -85,B 0,C 180,E1 -13845.971,E2 -13845.971} C_VEL
LIN {X 0,Y 347.934,Z 390.641,A -85,B 0,C 180,E1 -13849.526,E2 -13849.526} C_VEL
LIN {X 0,Y 348.084,Z 390.623,A -85,B 0,C 180,E1 -13853.042,E2 -13853.042} C_VEL
LIN {X 0,Y 348.209,Z 390.608,A -85,B 0,C 180,E1 -13857.687,E2 -13857.687} C_VEL
LIN {X 0,Y 348.347,Z 390.594,A -85,B 0,C 180,E1 -13860,E2 -13860} C_VEL
LIN {X 0,Y 348.211,Z 390.612,A -85,B 0,C 180,E1 -13862.314,E2 -13862.314} C_VEL
LIN {X 0,Y 348.109,Z 390.619,A -85,B 0,C 180,E1 -13866.958,E2 -13866.958} C_VEL
LIN {X 0,Y 347.97,Z 390.637,A -85,B 0,C 180,E1 -13869.299,E2 -13869.299} C_VEL
LIN {X 0,Y 347.892,Z 390.647,A -85,B 0,C 180,E1 -13872.839,E2 -13872.839} C_VEL
LIN {X 0,Y 347.842,Z 390.654,A -85,B 0,C 180,E1 -13876.431,E2 -13876.431} C_VEL
LIN {X 0,Y 347.862,Z 390.651,A -85,B 0,C 180,E1 -13878.86,E2 -13878.86} C_VEL
LIN {X 0,Y 347.779,Z 390.661,A -85,B 0,C 180,E1 -13882.579,E2 -13882.579} C_VEL
LIN {X 0,Y 347.814,Z 390.657,A -85,B 0,C 180,E1 -13885.108,E2 -13885.108} C_VEL
LIN {X 0,Y 347.814,Z 390.661,A -85,B 0,C 180,E1 -13887.694,E2 -13887.694} C_VEL
LIN {X 0,Y 347.766,Z 390.663,A -85,B 0,C 180,E1 -13890.346,E2 -13890.346} C_VEL
LIN {X 0,Y 347.746,Z 390.665,A -85,B 0,C 180,E1 -13894.464,E2 -13894.464} C_VEL
LIN {X 0,Y 347.779,Z 390.663,A -85,B 0,C 180,E1 -13897.99,E2 -13897.99} C_VEL
LIN {X 0,Y 347.758,Z 390.667,A -85,B 0,C 180,E1 -13901.829,E2 -13901.829} C_VEL
LIN {X 0,Y 347.709,Z 390.671,A -85,B 0,C 180,E1 -13905.027,E2 -13905.027} C_VEL
LIN {X 0,Y 347.752,Z 390.664,A -85,B 0,C 180,E1 -13908.397,E2 -13908.397} C_VEL
LIN {X 0,Y 347.776,Z 390.662,A -85,B 0,C 180,E1 -13912.011,E2 -13912.011} C_VEL
LIN {X 0,Y 347.746,Z 390.67,A -85,B 0,C 180,E1 -13915.536,E2 -13915.536} C_VEL
LIN {X 0,Y 347.766,Z 390.665,A -85,B 0,C 180,E1 -13919.654,E2 -13919.654} C_VEL
LIN {X 0,Y 347.88,Z 390.829,A -85,B 0,C 180,E1 -13923.08,E2 -13923.08} C_VEL
LIN {X 0,Y 349.786,Z 400.207,A -85,B 0,C 180,E1 -13925.992,E2 -13925.992} C_VEL
LIN {X 0,Y 350.474,Z 403.981,A -85,B 0,C 180,E1 -13927.055,E2 -13927.055} C_VEL
LIN {X 0,Y 353.482,Z 412.576,A -85,B 0,C 180,E1 -13927.449,E2 -13927.449} C_VEL
LIN {X 0,Y 357.344,Z 432.103,A -85,B 0,C 180,E1 -13928.123,E2 -13928.123} C_VEL
LIN {X 0,Y 356.042,Z 502.275,A -85,B 0,C 180,E1 -13929.528,E2 -13929.528} C_VEL
LIN {X 0,Y 355.702,Z 515.798,A -85,B 0,C 180,E1 -13929.885,E2 -13929.885} C_VEL
LIN {X 0,Y 354.934,Z 529.205,A -85,B 0,C 180,E1 -13930.48,E2 -13930.48} C_VEL
LIN {X 0,Y 354.116,Z 540.425,A -85,B 0,C 180,E1 -13931.185,E2 -13931.185} C_VEL
LIN {X 0,Y 353.074,Z 552.419,A -85,B 0,C 180,E1 -13932.179,E2 -13932.179} C_VEL
LIN {X 0,Y 351.969,Z 563.446,A -85,B 0,C 180,E1 -13933.364,E2 -13933.364} C_VEL
LIN {X 0,Y 350.985,Z 572.815,A -85,B 0,C 180,E1 -13934.615,E2 -13934.615} C_VEL
LIN {X 0,Y 349.843,Z 581.661,A -85,B 0,C 180,E1 -13936.051,E2 -13936.051} C_VEL
LIN {X 0,Y 348.736,Z 590.289,A -85,B 0,C 180,E1 -13937.784,E2 -13937.784} C_VEL
LIN {X 0,Y 347.863,Z 597.166,A -85,B 0,C 180,E1 -13939.524,E2 -13939.524} C_VEL
LIN {X 0,Y 347.172,Z 602.672,A -85,B 0,C 180,E1 -13941.267,E2 -13941.267} C_VEL
LIN {X 0,Y 346.632,Z 607.929,A -85,B 0,C 180,E1 -13943.456,E2 -13943.456} C_VEL
LIN {X 0,Y 346.414,Z 611.137,A -85,B 0,C 180,E1 -13945.345,E2 -13945.345} C_VEL
LIN {X 0,Y 346.24,Z 612.538,A -85,B 0,C 180,E1 -13946.509,E2 -13946.509} C_VEL
LIN {X 0,Y 346.137,Z 614.145,A -85,B 0,C 180,E1 -13948.837,E2 -13948.837} C_VEL
LIN {X 0,Y 346.119,Z 614.378,A -85,B 0,C 180,E1 -13950,E2 -13950} C_VEL
LIN {X 0,Y 346.136,Z 614.187,A -85,B 0,C 180,E1 -13951.164,E2 -13951.164} C_VEL
LIN {X 0,Y 346.238,Z 612.633,A -85,B 0,C 180,E1 -13953.491,E2 -13953.491} C_VEL
LIN {X 0,Y 346.408,Z 611.274,A -85,B 0,C 180,E1 -13954.655,E2 -13954.655} C_VEL
LIN {X 0,Y 346.629,Z 608.151,A -85,B 0,C 180,E1 -13956.539,E2 -13956.539} C_VEL
LIN {X 0,Y 346.995,Z 604.515,A -85,B 0,C 180,E1 -13958.151,E2 -13958.151} C_VEL
LIN {X 0,Y 347.563,Z 599.495,A -85,B 0,C 180,E1 -13959.897,E2 -13959.897} C_VEL
LIN {X 0,Y 348.333,Z 593.174,A -85,B 0,C 180,E1 -13961.64,E2 -13961.64} C_VEL
LIN {X 0,Y 349.352,Z 585.261,A -85,B 0,C 180,E1 -13963.377,E2 -13963.377} C_VEL
LIN {X 0,Y 350.657,Z 575.416,A -85,B 0,C 180,E1 -13965.103,E2 -13965.103} C_VEL
LIN {X 0,Y 351.758,Z 565.09,A -85,B 0,C 180,E1 -13966.541,E2 -13966.541} C_VEL
LIN {X 0,Y 352.834,Z 554.85,A -85,B 0,C 180,E1 -13967.684,E2 -13967.684} C_VEL
LIN {X 0,Y 353.907,Z 543.649,A -85,B 0,C 180,E1 -13968.676,E2 -13968.676} C_VEL
LIN {X 0,Y 354.905,Z 531.024,A -85,B 0,C 180,E1 -13969.522,E2 -13969.522} C_VEL
LIN {X 0,Y 355.545,Z 518.367,A -85,B 0,C 180,E1 -13970.125,E2 -13970.125} C_VEL
LIN {X 0,Y 356.08,Z 505.345,A -85,B 0,C 180,E1 -13970.508,E2 -13970.508} C_VEL
LIN {X 0,Y 356.95,Z 456.628,A -85,B 0,C 180,E1 -13971.487,E2 -13971.487} C_VEL
LIN {X 0,Y 356.467,Z 450.811,A -85,B 0,C 180,E1 -13971.641,E2 -13971.641} C_VEL
LIN {X 0,Y 354.036,Z 441.466,A -85,B 0,C 180,E1 -13971.999,E2 -13971.999} C_VEL
LIN {X 0,Y 351.58,Z 434.085,A -85,B 0,C 180,E1 -13972.322,E2 -13972.322} C_VEL
LIN {X 0,Y 349.596,Z 426.545,A -85,B 0,C 180,E1 -13972.621,E2 -13972.621} C_VEL
LIN {X 0,Y 346.734,Z 413.12,A -85,B 0,C 180,E1 -13973.115,E2 -13973.115} C_VEL
LIN {X 0,Y 343.284,Z 403.815,A -85,B 0,C 180,E1 -13973.588,E2 -13973.588} C_VEL
LIN {X 0,Y 341.15,Z 393.124,A -85,B 0,C 180,E1 -13976.951,E2 -13976.951} C_VEL
LIN {X 0,Y 340.791,Z 391.536,A -85,B 0,C 180,E1 -13977.529,E2 -13977.529} C_VEL
LIN {X 0,Y 340.707,Z 391.547,A -85,B 0,C 180,E1 -13981.044,E2 -13981.044} C_VEL
LIN {X 0,Y 340.721,Z 391.541,A -85,B 0,C 180,E1 -13985.279,E2 -13985.279} C_VEL
LIN {X 0,Y 340.713,Z 391.545,A -85,B 0,C 180,E1 -13988.386,E2 -13988.386} C_VEL
LIN {X 0,Y 340.702,Z 391.544,A -85,B 0,C 180,E1 -13992.046,E2 -13992.046} C_VEL
LIN {X 0,Y 340.686,Z 391.544,A -85,B 0,C 180,E1 -13995.461,E2 -13995.461} C_VEL
LIN {X 0,Y 340.697,Z 391.545,A -85,B 0,C 180,E1 -13998.692,E2 -13998.692} C_VEL
LIN {X 0,Y 340.74,Z 391.536,A -85,B 0,C 180,E1 -14001.773,E2 -14001.773} C_VEL
LIN {X 0,Y 340.727,Z 391.539,A -85,B 0,C 180,E1 -14005.596,E2 -14005.596} C_VEL
LIN {X 0,Y 340.708,Z 391.542,A -85,B 0,C 180,E1 -14008.956,E2 -14008.956} C_VEL
LIN {X 0,Y 340.784,Z 391.536,A -85,B 0,C 180,E1 -14012.474,E2 -14012.474} C_VEL
LIN {X 0,Y 340.76,Z 391.535,A -85,B 0,C 180,E1 -14015.639,E2 -14015.639} C_VEL
LIN {X 0,Y 340.77,Z 391.534,A -85,B 0,C 180,E1 -14019.475,E2 -14019.475} C_VEL
LIN {X 0,Y 340.863,Z 391.526,A -85,B 0,C 180,E1 -14021.984,E2 -14021.984} C_VEL
LIN {X 0,Y 340.874,Z 391.523,A -85,B 0,C 180,E1 -14025.705,E2 -14025.705} C_VEL
LIN {X 0,Y 340.876,Z 391.521,A -85,B 0,C 180,E1 -14029.306,E2 -14029.306} C_VEL
LIN {X 0,Y 341.081,Z 391.493,A -85,B 0,C 180,E1 -14032.898,E2 -14032.898} C_VEL
LIN {X 0,Y 341.173,Z 391.487,A -85,B 0,C 180,E1 -14037.639,E2 -14037.639} C_VEL
LIN {X 0,Y 341.3,Z 391.472,A -85,B 0,C 180,E1 -14040,E2 -14040} C_VEL
LIN {X 0,Y 341.173,Z 391.485,A -85,B 0,C 180,E1 -14042.361,E2 -14042.361} C_VEL
LIN {X 0,Y 341.054,Z 391.499,A -85,B 0,C 180,E1 -14047.102,E2 -14047.102} C_VEL
LIN {X 0,Y 340.878,Z 391.52,A -85,B 0,C 180,E1 -14050.694,E2 -14050.694} C_VEL
LIN {X 0,Y 340.867,Z 391.522,A -85,B 0,C 180,E1 -14054.325,E2 -14054.325} C_VEL
LIN {X 0,Y 340.841,Z 391.525,A -85,B 0,C 180,E1 -14058.466,E2 -14058.466} C_VEL
LIN {X 0,Y 340.758,Z 391.536,A -85,B 0,C 180,E1 -14061.857,E2 -14061.857} C_VEL
LIN {X 0,Y 340.776,Z 391.537,A -85,B 0,C 180,E1 -14065.664,E2 -14065.664} C_VEL
LIN {X 0,Y 340.732,Z 391.538,A -85,B 0,C 180,E1 -14068.32,E2 -14068.32} C_VEL
LIN {X 0,Y 340.701,Z 391.545,A -85,B 0,C 180,E1 -14071.044,E2 -14071.044} C_VEL
LIN {X 0,Y 340.721,Z 391.546,A -85,B 0,C 180,E1 -14075.279,E2 -14075.279} C_VEL
LIN {X 0,Y 340.713,Z 391.541,A -85,B 0,C 180,E1 -14078.386,E2 -14078.386} C_VEL
LIN {X 0,Y 340.702,Z 391.543,A -85,B 0,C 180,E1 -14082.045,E2 -14082.045} C_VEL
LIN {X 0,Y 340.686,Z 391.547,A -85,B 0,C 180,E1 -14085.461,E2 -14085.461} C_VEL
LIN {X 0,Y 340.689,Z 391.547,A -85,B 0,C 180,E1 -14088.69,E2 -14088.69} C_VEL
LIN {X 0,Y 340.736,Z 391.539,A -85,B 0,C 180,E1 -14091.772,E2 -14091.772} C_VEL
LIN {X 0,Y 340.726,Z 391.541,A -85,B 0,C 180,E1 -14095.595,E2 -14095.595} C_VEL
LIN {X 0,Y 340.743,Z 391.555,A -85,B 0,C 180,E1 -14099.092,E2 -14099.092} C_VEL
LIN {X 0,Y 343.092,Z 402.238,A -85,B 0,C 180,E1 -14102.223,E2 -14102.223} C_VEL
LIN {X 0,Y 344.913,Z 412.121,A -85,B 0,C 180,E1 -14104.988,E2 -14104.988} C_VEL
LIN {X 0,Y 344.325,Z 418.172,A -85,B 0,C 180,E1 -14106.531,E2 -14106.531} C_VEL
LIN {X 0,Y 349.187,Z 445.647,A -85,B 0,C 180,E1 -14107.482,E2 -14107.482} C_VEL
LIN {X 0,Y 350.466,Z 454.676,A -85,B 0,C 180,E1 -14107.763,E2 -14107.763} C_VEL
LIN {X 0,Y 349.029,Z 526.384,A -85,B 0,C 180,E1 -14109.251,E2 -14109.251} C_VEL
LIN {X 0,Y 348.315,Z 539.586,A -85,B 0,C 180,E1 -14109.747,E2 -14109.747} C_VEL
LIN {X 0,Y 347.251,Z 552.826,A -85,B 0,C 180,E1 -14110.491,E2 -14110.491} C_VEL
LIN {X 0,Y 346.189,Z 563.946,A -85,B 0,C 180,E1 -14111.352,E2 -14111.352} C_VEL
LIN {X 0,Y 344.906,Z 575.525,A -85,B 0,C 180,E1 -14112.509,E2 -14112.509} C_VEL
LIN {X 0,Y 343.707,Z 585.506,A -85,B 0,C 180,E1 -14113.76,E2 -14113.76} C_VEL
LIN {X 0,Y 342.639,Z 594.479,A -85,B 0,C 180,E1 -14115.144,E2 -14115.144} C_VEL
LIN {X 0,Y 341.679,Z 602.347,A -85,B 0,C 180,E1 -14116.62,E2 -14116.62} C_VEL
LIN {X 0,Y 340.61,Z 610.029,A -85,B 0,C 180,E1 -14118.394,E2 -14118.394} C_VEL
LIN {X 0,Y 339.83,Z 617.118,A -85,B 0,C 180,E1 -14120.476,E2 -14120.476} C_VEL
LIN {X 0,Y 339.407,Z 621.835,A -85,B 0,C 180,E1 -14122.265,E2 -14122.265} C_VEL
LIN {X 0,Y 339.111,Z 625.614,A -85,B 0,C 180,E1 -14124.15,E2 -14124.15} C_VEL
LIN {X 0,Y 339.061,Z 627.298,A -85,B 0,C 180,E1 -14125.244,E2 -14125.244} C_VEL
LIN {X 0,Y 339.06,Z 628.693,A -85,B 0,C 180,E1 -14126.435,E2 -14126.435} C_VEL
LIN {X 0,Y 338.993,Z 630.295,A -85,B 0,C 180,E1 -14128.812,E2 -14128.812} C_VEL
LIN {X 0,Y 339.017,Z 630.509,A -85,B 0,C 180,E1 -14130,E2 -14130} C_VEL
LIN {X 0,Y 338.993,Z 630.29,A -85,B 0,C 180,E1 -14131.188,E2 -14131.188} C_VEL
LIN {X 0,Y 339.06,Z 628.683,A -85,B 0,C 180,E1 -14133.565,E2 -14133.565} C_VEL
LIN {X 0,Y 339.062,Z 627.283,A -85,B 0,C 180,E1 -14134.756,E2 -14134.756} C_VEL
LIN {X 0,Y 339.176,Z 624.343,A -85,B 0,C 180,E1 -14136.544,E2 -14136.544} C_VEL
LIN {X 0,Y 339.536,Z 620.367,A -85,B 0,C 180,E1 -14138.331,E2 -14138.331} C_VEL
LIN {X 0,Y 340.128,Z 614.253,A -85,B 0,C 180,E1 -14140.416,E2 -14140.416} C_VEL
LIN {X 0,Y 340.918,Z 607.576,A -85,B 0,C 180,E1 -14142.199,E2 -14142.199} C_VEL
LIN {X 0,Y 342.09,Z 599.297,A -85,B 0,C 180,E1 -14143.969,E2 -14143.969} C_VEL
LIN {X 0,Y 343.165,Z 590.095,A -85,B 0,C 180,E1 -14145.552,E2 -14145.552} C_VEL
LIN {X 0,Y 344.418,Z 579.134,A -85,B 0,C 180,E1 -14147.057,E2 -14147.057} C_VEL
LIN {X 0,Y 345.675,Z 568.503,A -85,B 0,C 180,E1 -14148.215,E2 -14148.215} C_VEL
LIN {X 0,Y 346.855,Z 556.616,A -85,B 0,C 180,E1 -14149.224,E2 -14149.224} C_VEL
LIN {X 0,Y 347.934,Z 544.247,A -85,B 0,C 180,E1 -14150.006,E2 -14150.006} C_VEL
LIN {X 0,Y 348.767,Z 531.527,A -85,B 0,C 180,E1 -14150.572,E2 -14150.572} C_VEL
LIN {X 0,Y 349.286,Z 518.135,A -85,B 0,C 180,E1 -14150.925,E2 -14150.925} C_VEL
LIN {X 0,Y 350.298,Z 452.808,A -85,B 0,C 180,E1 -14152.271,E2 -14152.271} C_VEL
LIN {X 0,Y 345.732,Z 425.749,A -85,B 0,C 180,E1 -14153.176,E2 -14153.176} C_VEL
LIN {X 0,Y 344.309,Z 418.082,A -85,B 0,C 180,E1 -14153.474,E2 -14153.474} C_VEL
LIN {X 0,Y 344.897,Z 412.043,A -85,B 0,C 180,E1 -14155.013,E2 -14155.013} C_VEL
LIN {X 0,Y 342.803,Z 400.791,A -85,B 0,C 180,E1 -14158.168,E2 -14158.168} C_VEL
LIN {X 0,Y 340.745,Z 391.541,A -85,B 0,C 180,E1 -14160.907,E2 -14160.907} C_VEL
LIN {X 0,Y 340.719,Z 391.544,A -85,B 0,C 180,E1 -14165.279,E2 -14165.279} C_VEL
LIN {X 0,Y 340.711,Z 391.543,A -85,B 0,C 180,E1 -14168.386,E2 -14168.386} C_VEL
LIN {X 0,Y 340.7,Z 391.543,A -85,B 0,C 180,E1 -14172.045,E2 -14172.045} C_VEL
LIN {X 0,Y 340.684,Z 391.546,A -85,B 0,C 180,E1 -14175.461,E2 -14175.461} C_VEL
LIN {X 0,Y 340.688,Z 391.549,A -85,B 0,C 180,E1 -14178.691,E2 -14178.691} C_VEL
LIN {X 0,Y 340.734,Z 391.538,A -85,B 0,C 180,E1 -14181.773,E2 -14181.773} C_VEL
LIN {X 0,Y 340.724,Z 391.539,A -85,B 0,C 180,E1 -14185.595,E2 -14185.595} C_VEL
LIN {X 0,Y 340.699,Z 391.546,A -85,B 0,C 180,E1 -14188.955,E2 -14188.955} C_VEL
LIN {X 0,Y 340.805,Z 391.532,A -85,B 0,C 180,E1 -14193.02,E2 -14193.02} C_VEL
LIN {X 0,Y 340.731,Z 391.541,A -85,B 0,C 180,E1 -14196.927,E2 -14196.927} C_VEL
LIN {X 0,Y 340.793,Z 391.535,A -85,B 0,C 180,E1 -14200.734,E2 -14200.734} C_VEL
LIN {X 0,Y 340.789,Z 391.532,A -85,B 0,C 180,E1 -14203.219,E2 -14203.219} C_VEL
LIN {X 0,Y 340.849,Z 391.526,A -85,B 0,C 180,E1 -14206.891,E2 -14206.891} C_VEL
LIN {X 0,Y 340.914,Z 391.52,A -85,B 0,C 180,E1 -14210.507,E2 -14210.507} C_VEL
LIN {X 0,Y 341.051,Z 391.5,A -85,B 0,C 180,E1 -14212.898,E2 -14212.898} C_VEL
LIN {X 0,Y 341.17,Z 391.485,A -85,B 0,C 180,E1 -14217.639,E2 -14217.639} C_VEL
LIN {X 0,Y 341.297,Z 391.472,A -85,B 0,C 180,E1 -14220,E2 -14220} C_VEL
LIN {X 0,Y 341.173,Z 391.488,A -85,B 0,C 180,E1 -14222.361,E2 -14222.361} C_VEL
LIN {X 0,Y 341.078,Z 391.495,A -85,B 0,C 180,E1 -14227.102,E2 -14227.102} C_VEL
LIN {X 0,Y 340.873,Z 391.521,A -85,B 0,C 180,E1 -14230.694,E2 -14230.694} C_VEL
LIN {X 0,Y 340.865,Z 391.525,A -85,B 0,C 180,E1 -14234.325,E2 -14234.325} C_VEL
LIN {X 0,Y 340.841,Z 391.527,A -85,B 0,C 180,E1 -14238.467,E2 -14238.467} C_VEL
LIN {X 0,Y 340.755,Z 391.54,A -85,B 0,C 180,E1 -14241.857,E2 -14241.857} C_VEL
LIN {X 0,Y 340.775,Z 391.538,A -85,B 0,C 180,E1 -14245.664,E2 -14245.664} C_VEL
LIN {X 0,Y 340.744,Z 391.539,A -85,B 0,C 180,E1 -14248.32,E2 -14248.32} C_VEL
LIN {X 0,Y 340.706,Z 391.542,A -85,B 0,C 180,E1 -14251.044,E2 -14251.044} C_VEL
LIN {X 0,Y 340.72,Z 391.542,A -85,B 0,C 180,E1 -14255.279,E2 -14255.279} C_VEL
LIN {X 0,Y 340.715,Z 391.541,A -85,B 0,C 180,E1 -14258.387,E2 -14258.387} C_VEL
LIN {X 0,Y 340.705,Z 391.544,A -85,B 0,C 180,E1 -14262.046,E2 -14262.046} C_VEL
LIN {X 0,Y 340.654,Z 391.549,A -85,B 0,C 180,E1 -14266.227,E2 -14266.227} C_VEL
LIN {X 0,Y 340.69,Z 391.547,A -85,B 0,C 180,E1 -14269.753,E2 -14269.753} C_VEL
LIN {X 0,Y 340.707,Z 391.547,A -85,B 0,C 180,E1 -14273.259,E2 -14273.259} C_VEL
LIN {X 0,Y 340.696,Z 391.544,A -85,B 0,C 180,E1 -14276.154,E2 -14276.154} C_VEL
LIN {X 0,Y 340.776,Z 391.534,A -85,B 0,C 180,E1 -14280.333,E2 -14280.333} C_VEL
LIN {X 0,Y 340.827,Z 391.622,A -85,B 0,C 180,E1 -14282.67,E2 -14282.67} C_VEL
LIN {X 0,Y 342.841,Z 401.47,A -85,B 0,C 180,E1 -14285.796,E2 -14285.796} C_VEL
LIN {X 0,Y 343.33,Z 404.132,A -85,B 0,C 180,E1 -14286.548,E2 -14286.548} C_VEL
LIN {X 0,Y 347.218,Z 414.973,A -85,B 0,C 180,E1 -14287.068,E2 -14287.068} C_VEL
LIN {X 0,Y 350.789,Z 433.332,A -85,B 0,C 180,E1 -14287.715,E2 -14287.715} C_VEL
LIN {X 0,Y 349.418,Z 502.467,A -85,B 0,C 180,E1 -14289.122,E2 -14289.122} C_VEL
LIN {X 0,Y 349.049,Z 515.979,A -85,B 0,C 180,E1 -14289.484,E2 -14289.484} C_VEL
LIN {X 0,Y 348.266,Z 529.381,A -85,B 0,C 180,E1 -14290.09,E2 -14290.09} C_VEL
LIN {X 0,Y 347.419,Z 540.598,A -85,B 0,C 180,E1 -14290.809,E2 -14290.809} C_VEL
LIN {X 0,Y 346.334,Z 552.591,A -85,B 0,C 180,E1 -14291.82,E2 -14291.82} C_VEL
LIN {X 0,Y 345.16,Z 563.618,A -85,B 0,C 180,E1 -14293.027,E2 -14293.027} C_VEL
LIN {X 0,Y 344.145,Z 573.037,A -85,B 0,C 180,E1 -14294.309,E2 -14294.309} C_VEL
LIN {X 0,Y 342.967,Z 581.831,A -85,B 0,C 180,E1 -14295.765,E2 -14295.765} C_VEL
LIN {X 0,Y 341.792,Z 590.458,A -85,B 0,C 180,E1 -14297.532,E2 -14297.532} C_VEL
LIN {X 0,Y 340.847,Z 597.336,A -85,B 0,C 180,E1 -14299.306,E2 -14299.306} C_VEL
LIN {X 0,Y 340.135,Z 602.841,A -85,B 0,C 180,E1 -14301.085,E2 -14301.085} C_VEL
LIN {X 0,Y 339.674,Z 607.161,A -85,B 0,C 180,E1 -14302.869,E2 -14302.869} C_VEL
LIN {X 0,Y 339.474,Z 609.446,A -85,B 0,C 180,E1 -14304.059,E2 -14304.059} C_VEL
LIN {X 0,Y 339.334,Z 611.305,A -85,B 0,C 180,E1 -14305.248,E2 -14305.248} C_VEL
LIN {X 0,Y 339.169,Z 612.705,A -85,B 0,C 180,E1 -14306.436,E2 -14306.436} C_VEL
LIN {X 0,Y 339.04,Z 614.313,A -85,B 0,C 180,E1 -14308.812,E2 -14308.812} C_VEL
LIN {X 0,Y 339.022,Z 614.545,A -85,B 0,C 180,E1 -14310,E2 -14310} C_VEL
LIN {X 0,Y 339.039,Z 614.354,A -85,B 0,C 180,E1 -14311.188,E2 -14311.188} C_VEL
LIN {X 0,Y 339.167,Z 612.8,A -85,B 0,C 180,E1 -14313.564,E2 -14313.564} C_VEL
LIN {X 0,Y 339.328,Z 611.441,A -85,B 0,C 180,E1 -14314.752,E2 -14314.752} C_VEL
LIN {X 0,Y 339.545,Z 608.593,A -85,B 0,C 180,E1 -14316.525,E2 -14316.525} C_VEL
LIN {X 0,Y 339.957,Z 604.681,A -85,B 0,C 180,E1 -14318.321,E2 -14318.321} C_VEL
LIN {X 0,Y 340.562,Z 599.661,A -85,B 0,C 180,E1 -14320.103,E2 -14320.103} C_VEL
LIN {X 0,Y 341.386,Z 593.339,A -85,B 0,C 180,E1 -14321.881,E2 -14321.881} C_VEL
LIN {X 0,Y 342.427,Z 585.426,A -85,B 0,C 180,E1 -14323.652,E2 -14323.652} C_VEL
LIN {X 0,Y 343.795,Z 575.58,A -85,B 0,C 180,E1 -14325.412,E2 -14325.412} C_VEL
LIN {X 0,Y 344.774,Z 567.033,A -85,B 0,C 180,E1 -14326.65,E2 -14326.65} C_VEL
LIN {X 0,Y 345.927,Z 556.435,A -85,B 0,C 180,E1 -14327.896,E2 -14327.896} C_VEL
LIN {X 0,Y 347.032,Z 545.571,A -85,B 0,C 180,E1 -14328.907,E2 -14328.907} C_VEL
LIN {X 0,Y 348.086,Z 533.567,A -85,B 0,C 180,E1 -14329.767,E2 -14329.767} C_VEL
LIN {X 0,Y 348.792,Z 521.246,A -85,B 0,C 180,E1 -14330.417,E2 -14330.417} C_VEL
LIN {X 0,Y 349.357,Z 508.5,A -85,B 0,C 180,E1 -14330.844,E2 -14330.844} C_VEL
LIN {X 0,Y 350.745,Z 432.648,A -85,B 0,C 180,E1 -14332.409,E2 -14332.409} C_VEL
LIN {X 0,Y 349.596,Z 426.545,A -85,B 0,C 180,E1 -14332.621,E2 -14332.621} C_VEL
LIN {X 0,Y 348.217,Z 423.003,A -85,B 0,C 180,E1 -14332.794,E2 -14332.794} C_VEL
LIN {X 0,Y 344.276,Z 418.108,A -85,B 0,C 180,E1 -14333.18,E2 -14333.18} C_VEL
LIN {X 0,Y 340.098,Z 413.314,A -85,B 0,C 180,E1 -14333.592,E2 -14333.592} C_VEL
LIN {X 0,Y 338.359,Z 409.892,A -85,B 0,C 180,E1 -14333.8,E2 -14333.8} C_VEL
LIN {X 0,Y 336.115,Z 403.974,A -85,B 0,C 180,E1 -14334.127,E2 -14334.127} C_VEL
LIN {X 0,Y 333.922,Z 393.291,A -85,B 0,C 180,E1 -14337.583,E2 -14337.583} C_VEL
LIN {X 0,Y 333.716,Z 392.419,A -85,B 0,C 180,E1 -14337.926,E2 -14337.926} C_VEL
LIN {X 0,Y 333.7,Z 392.419,A -85,B 0,C 180,E1 -14340.362,E2 -14340.362} C_VEL
LIN {X 0,Y 333.689,Z 392.422,A -85,B 0,C 180,E1 -14344.774,E2 -14344.774} C_VEL
LIN {X 0,Y 333.655,Z 392.421,A -85,B 0,C 180,E1 -14347.651,E2 -14347.651} C_VEL
LIN {X 0,Y 333.65,Z 392.426,A -85,B 0,C 180,E1 -14350.768,E2 -14350.768} C_VEL
LIN {X 0,Y 333.63,Z 392.426,A -85,B 0,C 180,E1 -14354.257,E2 -14354.257} C_VEL
LIN {X 0,Y 333.648,Z 392.422,A -85,B 0,C 180,E1 -14357.619,E2 -14357.619} C_VEL
LIN {X 0,Y 333.659,Z 392.418,A -85,B 0,C 180,E1 -14361.202,E2 -14361.202} C_VEL
LIN {X 0,Y 333.681,Z 392.418,A -85,B 0,C 180,E1 -14363.861,E2 -14363.861} C_VEL
LIN {X 0,Y 333.649,Z 392.421,A -85,B 0,C 180,E1 -14367.413,E2 -14367.413} C_VEL
LIN {X 0,Y 333.716,Z 392.413,A -85,B 0,C 180,E1 -14371.028,E2 -14371.028} C_VEL
LIN {X 0,Y 333.74,Z 392.411,A -85,B 0,C 180,E1 -14373.754,E2 -14373.754} C_VEL
LIN {X 0,Y 333.724,Z 392.415,A -85,B 0,C 180,E1 -14377.914,E2 -14377.914} C_VEL
LIN {X 0,Y 333.8,Z 392.402,A -85,B 0,C 180,E1 -14381.59,E2 -14381.59} C_VEL
LIN {X 0,Y 333.813,Z 392.402,A -85,B 0,C 180,E1 -14385.577,E2 -14385.577} C_VEL
LIN {X 0,Y 333.838,Z 392.398,A -85,B 0,C 180,E1 -14389.078,E2 -14389.078} C_VEL
LIN {X 0,Y 334.031,Z 392.371,A -85,B 0,C 180,E1 -14392.748,E2 -14392.748} C_VEL
LIN {X 0,Y 333.816,Z 392.4,A -85,B 0,C 180,E1 -14395.169,E2 -14395.169} C_VEL
LIN {X 0,Y 334.111,Z 392.367,A -85,B 0,C 180,E1 -14397.589,E2 -14397.589} C_VEL
LIN {X 0,Y 334.251,Z 392.35,A -85,B 0,C 180,E1 -14400,E2 -14400} C_VEL
LIN {X 0,Y 334.111,Z 392.365,A -85,B 0,C 180,E1 -14402.411,E2 -14402.411} C_VEL
LIN {X 0,Y 334.015,Z 392.377,A -85,B 0,C 180,E1 -14406.039,E2 -14406.039} C_VEL
LIN {X 0,Y 333.855,Z 392.4,A -85,B 0,C 180,E1 -14409.695,E2 -14409.695} C_VEL
LIN {X 0,Y 333.803,Z 392.405,A -85,B 0,C 180,E1 -14413.391,E2 -14413.391} C_VEL
LIN {X 0,Y 333.751,Z 392.409,A -85,B 0,C 180,E1 -14417.146,E2 -14417.146} C_VEL
LIN {X 0,Y 333.743,Z 392.414,A -85,B 0,C 180,E1 -14419.69,E2 -14419.69} C_VEL
LIN {X 0,Y 333.696,Z 392.414,A -85,B 0,C 180,E1 -14422.278,E2 -14422.278} C_VEL
LIN {X 0,Y 333.739,Z 392.41,A -85,B 0,C 180,E1 -14426.246,E2 -14426.246} C_VEL
LIN {X 0,Y 333.694,Z 392.418,A -85,B 0,C 180,E1 -14428.974,E2 -14428.974} C_VEL
LIN {X 0,Y 333.647,Z 392.422,A -85,B 0,C 180,E1 -14432.587,E2 -14432.587} C_VEL
LIN {X 0,Y 333.679,Z 392.417,A -85,B 0,C 180,E1 -14436.139,E2 -14436.139} C_VEL
LIN {X 0,Y 333.65,Z 392.427,A -85,B 0,C 180,E1 -14439.192,E2 -14439.192} C_VEL
LIN {X 0,Y 333.636,Z 392.424,A -85,B 0,C 180,E1 -14442.5,E2 -14442.5} C_VEL
LIN {X 0,Y 333.624,Z 392.425,A -85,B 0,C 180,E1 -14445.959,E2 -14445.959} C_VEL
LIN {X 0,Y 333.65,Z 392.425,A -85,B 0,C 180,E1 -14449.315,E2 -14449.315} C_VEL
LIN {X 0,Y 333.668,Z 392.424,A -85,B 0,C 180,E1 -14453.167,E2 -14453.167} C_VEL
LIN {X 0,Y 333.677,Z 392.421,A -85,B 0,C 180,E1 -14455.341,E2 -14455.341} C_VEL
LIN {X 0,Y 333.684,Z 392.46,A -85,B 0,C 180,E1 -14458.67,E2 -14458.67} C_VEL
LIN {X 0,Y 336.146,Z 403.599,A -85,B 0,C 180,E1 -14462.018,E2 -14462.018} C_VEL
LIN {X 0,Y 337.953,Z 413.181,A -85,B 0,C 180,E1 -14464.766,E2 -14464.766} C_VEL
LIN {X 0,Y 337.561,Z 417.992,A -85,B 0,C 180,E1 -14466.027,E2 -14466.027} C_VEL
LIN {X 0,Y 342.532,Z 445.679,A -85,B 0,C 180,E1 -14467.023,E2 -14467.023} C_VEL
LIN {X 0,Y 343.878,Z 455.887,A -85,B 0,C 180,E1 -14467.344,E2 -14467.344} C_VEL
LIN {X 0,Y 342.4,Z 526.23,A -85,B 0,C 180,E1 -14468.83,E2 -14468.83} C_VEL
LIN {X 0,Y 341.653,Z 539.428,A -85,B 0,C 180,E1 -14469.334,E2 -14469.334} C_VEL
LIN {X 0,Y 340.651,Z 551.549,A -85,B 0,C 180,E1 -14470.019,E2 -14470.019} C_VEL
LIN {X 0,Y 339.457,Z 563.783,A -85,B 0,C 180,E1 -14470.968,E2 -14470.968} C_VEL
LIN {X 0,Y 338.117,Z 575.361,A -85,B 0,C 180,E1 -14472.146,E2 -14472.146} C_VEL
LIN {X 0,Y 336.827,Z 585.751,A -85,B 0,C 180,E1 -14473.478,E2 -14473.478} C_VEL
LIN {X 0,Y 335.755,Z 594.314,A -85,B 0,C 180,E1 -14474.832,E2 -14474.832} C_VEL
LIN {X 0,Y 334.753,Z 602.182,A -85,B 0,C 180,E1 -14476.338,E2 -14476.338} C_VEL
LIN {X 0,Y 333.632,Z 609.863,A -85,B 0,C 180,E1 -14478.148,E2 -14478.148} C_VEL
LIN {X 0,Y 332.804,Z 616.951,A -85,B 0,C 180,E1 -14480.273,E2 -14480.273} C_VEL
LIN {X 0,Y 332.364,Z 621.668,A -85,B 0,C 180,E1 -14482.1,E2 -14482.1} C_VEL
LIN {X 0,Y 332.006,Z 625.774,A -85,B 0,C 180,E1 -14484.218,E2 -14484.218} C_VEL
LIN {X 0,Y 331.964,Z 628.526,A -85,B 0,C 180,E1 -14486.358,E2 -14486.358} C_VEL
LIN {X 0,Y 331.9,Z 630.128,A -85,B 0,C 180,E1 -14488.786,E2 -14488.786} C_VEL
LIN {X 0,Y 331.921,Z 630.342,A -85,B 0,C 180,E1 -14490,E2 -14490} C_VEL
LIN {X 0,Y 331.9,Z 630.122,A -85,B 0,C 180,E1 -14491.213,E2 -14491.213} C_VEL
LIN {X 0,Y 331.964,Z 628.516,A -85,B 0,C 180,E1 -14493.641,E2 -14493.641} C_VEL
LIN {X 0,Y 332.006,Z 625.753,A -85,B 0,C 180,E1 -14495.781,E2 -14495.781} C_VEL
LIN {X 0,Y 332.363,Z 621.632,A -85,B 0,C 180,E1 -14497.9,E2 -14497.9} C_VEL
LIN {X 0,Y 332.803,Z 616.905,A -85,B 0,C 180,E1 -14499.726,E2 -14499.726} C_VEL
LIN {X 0,Y 333.626,Z 609.807,A -85,B 0,C 180,E1 -14501.852,E2 -14501.852} C_VEL
LIN {X 0,Y 334.748,Z 602.106,A -85,B 0,C 180,E1 -14503.662,E2 -14503.662} C_VEL
LIN {X 0,Y 335.991,Z 592.435,A -85,B 0,C 180,E1 -14505.468,E2 -14505.468} C_VEL
LIN {X 0,Y 337.204,Z 582.457,A -85,B 0,C 180,E1 -14506.965,E2 -14506.965} C_VEL
LIN {X 0,Y 338.575,Z 571.188,A -85,B 0,C 180,E1 -14508.298,E2 -14508.298} C_VEL
LIN {X 0,Y 339.804,Z 560.147,A -85,B 0,C 180,E1 -14509.324,E2 -14509.324} C_VEL
LIN {X 0,Y 340.987,Z 547.904,A -85,B 0,C 180,E1 -14510.196,E2 -14510.196} C_VEL
LIN {X 0,Y 341.854,Z 535.93,A -85,B 0,C 180,E1 -14510.81,E2 -14510.81} C_VEL
LIN {X 0,Y 342.555,Z 522.808,A -85,B 0,C 180,E1 -14511.238,E2 -14511.238} C_VEL
LIN {X 0,Y 343.746,Z 453.883,A -85,B 0,C 180,E1 -14512.691,E2 -14512.691} C_VEL
LIN {X 0,Y 339.202,Z 426.943,A -85,B 0,C 180,E1 -14513.617,E2 -14513.617} C_VEL
LIN {X 0,Y 337.548,Z 417.989,A -85,B 0,C 180,E1 -14513.952,E2 -14513.952} C_VEL
LIN {X 0,Y 337.937,Z 413.096,A -85,B 0,C 180,E1 -14515.235,E2 -14515.235} C_VEL
LIN {X 0,Y 335.8,Z 401.829,A -85,B 0,C 180,E1 -14518.475,E2 -14518.475} C_VEL
LIN {X 0,Y 333.668,Z 392.424,A -85,B 0,C 180,E1 -14521.331,E2 -14521.331} C_VEL
LIN {X 0,Y 333.687,Z 392.42,A -85,B 0,C 180,E1 -14524.774,E2 -14524.774} C_VEL
LIN {X 0,Y 333.653,Z 392.422,A -85,B 0,C 180,E1 -14527.651,E2 -14527.651} C_VEL
LIN {X 0,Y 333.648,Z 392.425,A -85,B 0,C 180,E1 -14530.767,E2 -14530.767} C_VEL
LIN {X 0,Y 333.626,Z 392.424,A -85,B 0,C 180,E1 -14534.256,E2 -14534.256} C_VEL
LIN {X 0,Y 333.644,Z 392.422,A -85,B 0,C 180,E1 -14537.619,E2 -14537.619} C_VEL
LIN {X 0,Y 333.654,Z 392.422,A -85,B 0,C 180,E1 -14541.202,E2 -14541.202} C_VEL
LIN {X 0,Y 333.677,Z 392.417,A -85,B 0,C 180,E1 -14543.861,E2 -14543.861} C_VEL
LIN {X 0,Y 333.645,Z 392.422,A -85,B 0,C 180,E1 -14547.413,E2 -14547.413} C_VEL
LIN {X 0,Y 333.691,Z 392.418,A -85,B 0,C 180,E1 -14551.026,E2 -14551.026} C_VEL
LIN {X 0,Y 333.736,Z 392.41,A -85,B 0,C 180,E1 -14553.754,E2 -14553.754} C_VEL
LIN {X 0,Y 333.721,Z 392.413,A -85,B 0,C 180,E1 -14557.914,E2 -14557.914} C_VEL
LIN {X 0,Y 333.795,Z 392.402,A -85,B 0,C 180,E1 -14561.59,E2 -14561.59} C_VEL
LIN {X 0,Y 333.81,Z 392.4,A -85,B 0,C 180,E1 -14565.577,E2 -14565.577} C_VEL
LIN {X 0,Y 333.839,Z 392.397,A -85,B 0,C 180,E1 -14569.078,E2 -14569.078} C_VEL
LIN {X 0,Y 333.997,Z 392.38,A -85,B 0,C 180,E1 -14572.747,E2 -14572.747} C_VEL
LIN {X 0,Y 333.81,Z 392.4,A -85,B 0,C 180,E1 -14575.169,E2 -14575.169} C_VEL
LIN {X 0,Y 334.108,Z 392.364,A -85,B 0,C 180,E1 -14577.589,E2 -14577.589} C_VEL
LIN {X 0,Y 334.248,Z 392.35,A -85,B 0,C 180,E1 -14580,E2 -14580} C_VEL
LIN {X 0,Y 334.11,Z 392.367,A -85,B 0,C 180,E1 -14582.411,E2 -14582.411} C_VEL
LIN {X 0,Y 334.028,Z 392.373,A -85,B 0,C 180,E1 -14587.253,E2 -14587.253} C_VEL
LIN {X 0,Y 333.836,Z 392.397,A -85,B 0,C 180,E1 -14590.922,E2 -14590.922} C_VEL
LIN {X 0,Y 333.81,Z 392.402,A -85,B 0,C 180,E1 -14594.634,E2 -14594.634} C_VEL
LIN {X 0,Y 333.8,Z 392.403,A -85,B 0,C 180,E1 -14598.656,E2 -14598.656} C_VEL
LIN {X 0,Y 333.694,Z 392.417,A -85,B 0,C 180,E1 -14602.278,E2 -14602.278} C_VEL
LIN {X 0,Y 333.738,Z 392.411,A -85,B 0,C 180,E1 -14606.246,E2 -14606.246} C_VEL
LIN {X 0,Y 333.713,Z 392.413,A -85,B 0,C 180,E1 -14608.972,E2 -14608.972} C_VEL
LIN {X 0,Y 333.647,Z 392.421,A -85,B 0,C 180,E1 -14612.588,E2 -14612.588} C_VEL
LIN {X 0,Y 333.679,Z 392.419,A -85,B 0,C 180,E1 -14616.139,E2 -14616.139} C_VEL
LIN {X 0,Y 333.67,Z 392.42,A -85,B 0,C 180,E1 -14619.189,E2 -14619.189} C_VEL
LIN {X 0,Y 333.637,Z 392.423,A -85,B 0,C 180,E1 -14622.501,E2 -14622.501} C_VEL
LIN {X 0,Y 333.598,Z 392.429,A -85,B 0,C 180,E1 -14625.955,E2 -14625.955} C_VEL
LIN {X 0,Y 333.649,Z 392.426,A -85,B 0,C 180,E1 -14629.315,E2 -14629.315} C_VEL
LIN {X 0,Y 333.667,Z 392.423,A -85,B 0,C 180,E1 -14633.168,E2 -14633.168} C_VEL
LIN {X 0,Y 333.64,Z 392.424,A -85,B 0,C 180,E1 -14636.792,E2 -14636.792} C_VEL
LIN {X 0,Y 333.704,Z 392.416,A -85,B 0,C 180,E1 -14639.71,E2 -14639.71} C_VEL
LIN {X 0,Y 333.743,Z 392.469,A -85,B 0,C 180,E1 -14642.256,E2 -14642.256} C_VEL
LIN {X 0,Y 335.655,Z 401.647,A -85,B 0,C 180,E1 -14645.244,E2 -14645.244} C_VEL
LIN {X 0,Y 336.135,Z 404.135,A -85,B 0,C 180,E1 -14646.01,E2 -14646.01} C_VEL
LIN {X 0,Y 340.824,Z 416.772,A -85,B 0,C 180,E1 -14646.648,E2 -14646.648} C_VEL
LIN {X 0,Y 344.238,Z 434.089,A -85,B 0,C 180,E1 -14647.28,E2 -14647.28} C_VEL
LIN {X 0,Y 342.818,Z 502.658,A -85,B 0,C 180,E1 -14648.7,E2 -14648.7} C_VEL
LIN {X 0,Y 342.414,Z 516.16,A -85,B 0,C 180,E1 -14649.068,E2 -14649.068} C_VEL
LIN {X 0,Y 341.609,Z 529.557,A -85,B 0,C 180,E1 -14649.686,E2 -14649.686} C_VEL
LIN {X 0,Y 340.719,Z 540.773,A -85,B 0,C 180,E1 -14650.416,E2 -14650.416} C_VEL
LIN {X 0,Y 339.605,Z 552.763,A -85,B 0,C 180,E1 -14651.447,E2 -14651.447} C_VEL
LIN {X 0,Y 338.386,Z 563.789,A -85,B 0,C 180,E1 -14652.676,E2 -14652.676} C_VEL
LIN {X 0,Y 337.297,Z 573.376,A -85,B 0,C 180,E1 -14654.009,E2 -14654.009} C_VEL
LIN {X 0,Y 336.098,Z 582,A -85,B 0,C 180,E1 -14655.468,E2 -14655.468} C_VEL
LIN {X 0,Y 334.831,Z 590.628,A -85,B 0,C 180,E1 -14657.268,E2 -14657.268} C_VEL
LIN {X 0,Y 333.864,Z 597.505,A -85,B 0,C 180,E1 -14659.079,E2 -14659.079} C_VEL
LIN {X 0,Y 333.116,Z 603.01,A -85,B 0,C 180,E1 -14660.896,E2 -14660.896} C_VEL
LIN {X 0,Y 332.625,Z 607.329,A -85,B 0,C 180,E1 -14662.717,E2 -14662.717} C_VEL
LIN {X 0,Y 332.395,Z 609.615,A -85,B 0,C 180,E1 -14663.932,E2 -14663.932} C_VEL
LIN {X 0,Y 332.257,Z 611.473,A -85,B 0,C 180,E1 -14665.147,E2 -14665.147} C_VEL
LIN {X 0,Y 332.1,Z 612.872,A -85,B 0,C 180,E1 -14666.36,E2 -14666.36} C_VEL
LIN {X 0,Y 331.946,Z 614.48,A -85,B 0,C 180,E1 -14668.787,E2 -14668.787} C_VEL
LIN {X 0,Y 331.926,Z 614.712,A -85,B 0,C 180,E1 -14670,E2 -14670} C_VEL
LIN {X 0,Y 331.945,Z 614.521,A -85,B 0,C 180,E1 -14671.213,E2 -14671.213} C_VEL
LIN {X 0,Y 332.097,Z 612.966,A -85,B 0,C 180,E1 -14673.64,E2 -14673.64} C_VEL
LIN {X 0,Y 332.251,Z 611.607,A -85,B 0,C 180,E1 -14674.854,E2 -14674.854} C_VEL
LIN {X 0,Y 332.445,Z 609.071,A -85,B 0,C 180,E1 -14676.486,E2 -14676.486} C_VEL
LIN {X 0,Y 332.91,Z 604.848,A -85,B 0,C 180,E1 -14678.498,E2 -14678.498} C_VEL
LIN {X 0,Y 333.571,Z 599.826,A -85,B 0,C 180,E1 -14680.317,E2 -14680.317} C_VEL
LIN {X 0,Y 334.446,Z 593.504,A -85,B 0,C 180,E1 -14682.131,E2 -14682.131} C_VEL
LIN {X 0,Y 335.525,Z 585.591,A -85,B 0,C 180,E1 -14683.939,E2 -14683.939} C_VEL
LIN {X 0,Y 336.948,Z 575.744,A -85,B 0,C 180,E1 -14685.733,E2 -14685.733} C_VEL
LIN {X 0,Y 338.042,Z 566.581,A -85,B 0,C 180,E1 -14687.078,E2 -14687.078} C_VEL
LIN {X 0,Y 339.188,Z 556.597,A -85,B 0,C 180,E1 -14688.264,E2 -14688.264} C_VEL
LIN {X 0,Y 340.347,Z 545.732,A -85,B 0,C 180,E1 -14689.293,E2 -14689.293} C_VEL
LIN {X 0,Y 341.41,Z 533.726,A -85,B 0,C 180,E1 -14690.17,E2 -14690.17} C_VEL
LIN {X 0,Y 342.161,Z 521.401,A -85,B 0,C 180,E1 -14690.831,E2 -14690.831} C_VEL
LIN {X 0,Y 342.757,Z 508.645,A -85,B 0,C 180,E1 -14691.265,E2 -14691.265} C_VEL
LIN {X 0,Y 344.158,Z 434.236,A -85,B 0,C 180,E1 -14692.83,E2 -14692.83} C_VEL
LIN {X 0,Y 340.753,Z 416.233,A -85,B 0,C 180,E1 -14693.478,E2 -14693.478} C_VEL
LIN {X 0,Y 338.359,Z 409.892,A -85,B 0,C 180,E1 -14693.8,E2 -14693.8} C_VEL
LIN {X 0,Y 336.984,Z 406.796,A -85,B 0,C 180,E1 -14694.055,E2 -14694.055} C_VEL
LIN {X 0,Y 334.852,Z 403.817,A -85,B 0,C 180,E1 -14694.561,E2 -14694.561} C_VEL
LIN {X 0,Y 331.798,Z 400.798,A -85,B 0,C 180,E1 -14695.461,E2 -14695.461} C_VEL
LIN {X 0,Y 328.653,Z 397.693,A -85,B 0,C 180,E1 -14696.715,E2 -14696.715} C_VEL
LIN {X 0,Y 327.134,Z 395.055,A -85,B 0,C 180,E1 -14697.697,E2 -14697.697} C_VEL
LIN {X 0,Y 326.848,Z 394.103,A -85,B 0,C 180,E1 -14698.027,E2 -14698.027} C_VEL
LIN {X 0,Y 326.668,Z 393.296,A -85,B 0,C 180,E1 -14698.337,E2 -14698.337} C_VEL
LIN {X 0,Y 326.597,Z 393.305,A -85,B 0,C 180,E1 -14701.095,E2 -14701.095} C_VEL
LIN {X 0,Y 326.61,Z 393.3,A -85,B 0,C 180,E1 -14704.02,E2 -14704.02} C_VEL
LIN {X 0,Y 326.631,Z 393.298,A -85,B 0,C 180,E1 -14707.239,E2 -14707.239} C_VEL
LIN {X 0,Y 326.581,Z 393.304,A -85,B 0,C 180,E1 -14711.132,E2 -14711.132} C_VEL
LIN {X 0,Y 326.56,Z 393.308,A -85,B 0,C 180,E1 -14714.748,E2 -14714.748} C_VEL
LIN {X 0,Y 326.583,Z 393.304,A -85,B 0,C 180,E1 -14718.155,E2 -14718.155} C_VEL
LIN {X 0,Y 326.63,Z 393.292,A -85,B 0,C 180,E1 -14721.392,E2 -14721.392} C_VEL
LIN {X 0,Y 326.624,Z 393.297,A -85,B 0,C 180,E1 -14724.851,E2 -14724.851} C_VEL
LIN {X 0,Y 326.614,Z 393.298,A -85,B 0,C 180,E1 -14727.456,E2 -14727.456} C_VEL
LIN {X 0,Y 326.665,Z 393.295,A -85,B 0,C 180,E1 -14730.341,E2 -14730.341} C_VEL
LIN {X 0,Y 326.694,Z 393.288,A -85,B 0,C 180,E1 -14734.516,E2 -14734.516} C_VEL
LIN {X 0,Y 326.657,Z 393.294,A -85,B 0,C 180,E1 -14738.546,E2 -14738.546} C_VEL
LIN {X 0,Y 326.748,Z 393.279,A -85,B 0,C 180,E1 -14741.178,E2 -14741.178} C_VEL
LIN {X 0,Y 326.767,Z 393.278,A -85,B 0,C 180,E1 -14745.433,E2 -14745.433} C_VEL
LIN {X 0,Y 326.774,Z 393.278,A -85,B 0,C 180,E1 -14748.839,E2 -14748.839} C_VEL
LIN {X 0,Y 326.984,Z 393.249,A -85,B 0,C 180,E1 -14752.59,E2 -14752.59} C_VEL
LIN {X 0,Y 326.783,Z 393.276,A -85,B 0,C 180,E1 -14755.065,E2 -14755.065} C_VEL
LIN {X 0,Y 327.051,Z 393.246,A -85,B 0,C 180,E1 -14757.537,E2 -14757.537} C_VEL
LIN {X 0,Y 327.202,Z 393.228,A -85,B 0,C 180,E1 -14760,E2 -14760} C_VEL
LIN {X 0,Y 327.051,Z 393.244,A -85,B 0,C 180,E1 -14762.463,E2 -14762.463} C_VEL
LIN {X 0,Y 326.989,Z 393.251,A -85,B 0,C 180,E1 -14766.169,E2 -14766.169} C_VEL
LIN {X 0,Y 326.81,Z 393.275,A -85,B 0,C 180,E1 -14769.906,E2 -14769.906} C_VEL
LIN {X 0,Y 326.765,Z 393.284,A -85,B 0,C 180,E1 -14773.685,E2 -14773.685} C_VEL
LIN {X 0,Y 326.704,Z 393.289,A -85,B 0,C 180,E1 -14777.528,E2 -14777.528} C_VEL
LIN {X 0,Y 326.67,Z 393.291,A -85,B 0,C 180,E1 -14780.135,E2 -14780.135} C_VEL
LIN {X 0,Y 326.657,Z 393.293,A -85,B 0,C 180,E1 -14784.129,E2 -14784.129} C_VEL
LIN {X 0,Y 326.687,Z 393.29,A -85,B 0,C 180,E1 -14786.858,E2 -14786.858} C_VEL
LIN {X 0,Y 326.637,Z 393.295,A -85,B 0,C 180,E1 -14790.609,E2 -14790.609} C_VEL
LIN {X 0,Y 326.61,Z 393.298,A -85,B 0,C 180,E1 -14794.019,E2 -14794.019} C_VEL
LIN {X 0,Y 326.63,Z 393.301,A -85,B 0,C 180,E1 -14797.238,E2 -14797.238} C_VEL
LIN {X 0,Y 326.581,Z 393.307,A -85,B 0,C 180,E1 -14801.131,E2 -14801.131} C_VEL
LIN {X 0,Y 326.559,Z 393.307,A -85,B 0,C 180,E1 -14804.748,E2 -14804.748} C_VEL
LIN {X 0,Y 326.579,Z 393.303,A -85,B 0,C 180,E1 -14808.154,E2 -14808.154} C_VEL
LIN {X 0,Y 326.626,Z 393.299,A -85,B 0,C 180,E1 -14811.391,E2 -14811.391} C_VEL
LIN {X 0,Y 326.622,Z 393.3,A -85,B 0,C 180,E1 -14814.851,E2 -14814.851} C_VEL
LIN {X 0,Y 326.613,Z 393.367,A -85,B 0,C 180,E1 -14818.229,E2 -14818.229} C_VEL
LIN {X 0,Y 328.979,Z 403.679,A -85,B 0,C 180,E1 -14821.424,E2 -14821.424} C_VEL
LIN {X 0,Y 330.996,Z 414.236,A -85,B 0,C 180,E1 -14824.534,E2 -14824.534} C_VEL
LIN {X 0,Y 330.807,Z 417.847,A -85,B 0,C 180,E1 -14825.513,E2 -14825.513} C_VEL
LIN {X 0,Y 335.97,Z 446.434,A -85,B 0,C 180,E1 -14826.569,E2 -14826.569} C_VEL
LIN {X 0,Y 337.328,Z 455.422,A -85,B 0,C 180,E1 -14826.872,E2 -14826.872} C_VEL
LIN {X 0,Y 335.784,Z 526.076,A -85,B 0,C 180,E1 -14828.393,E2 -14828.393} C_VEL
LIN {X 0,Y 335.016,Z 539.269,A -85,B 0,C 180,E1 -14828.905,E2 -14828.905} C_VEL
LIN {X 0,Y 334.004,Z 551.388,A -85,B 0,C 180,E1 -14829.604,E2 -14829.604} C_VEL
LIN {X 0,Y 332.745,Z 563.621,A -85,B 0,C 180,E1 -14830.569,E2 -14830.569} C_VEL
LIN {X 0,Y 331.37,Z 575.198,A -85,B 0,C 180,E1 -14831.77,E2 -14831.77} C_VEL
LIN {X 0,Y 329.942,Z 585.944,A -85,B 0,C 180,E1 -14833.176,E2 -14833.176} C_VEL
LIN {X 0,Y 328.648,Z 595.823,A -85,B 0,C 180,E1 -14834.813,E2 -14834.813} C_VEL
LIN {X 0,Y 327.426,Z 604.75,A -85,B 0,C 180,E1 -14836.659,E2 -14836.659} C_VEL
LIN {X 0,Y 326.38,Z 611.934,A -85,B 0,C 180,E1 -14838.511,E2 -14838.511} C_VEL
LIN {X 0,Y 325.597,Z 618.479,A -85,B 0,C 180,E1 -14840.683,E2 -14840.683} C_VEL
LIN {X 0,Y 325.159,Z 622.811,A -85,B 0,C 180,E1 -14842.548,E2 -14842.548} C_VEL
LIN {X 0,Y 324.909,Z 625.874,A -85,B 0,C 180,E1 -14844.276,E2 -14844.276} C_VEL
LIN {X 0,Y 324.871,Z 628.359,A -85,B 0,C 180,E1 -14846.279,E2 -14846.279} C_VEL
LIN {X 0,Y 324.83,Z 629.354,A -85,B 0,C 180,E1 -14847.52,E2 -14847.52} C_VEL
LIN {X 0,Y 324.81,Z 629.961,A -85,B 0,C 180,E1 -14848.76,E2 -14848.76} C_VEL
LIN {X 0,Y 324.828,Z 630.175,A -85,B 0,C 180,E1 -14850,E2 -14850} C_VEL
LIN {X 0,Y 324.81,Z 629.955,A -85,B 0,C 180,E1 -14851.24,E2 -14851.24} C_VEL
LIN {X 0,Y 324.83,Z 629.346,A -85,B 0,C 180,E1 -14852.48,E2 -14852.48} C_VEL
LIN {X 0,Y 324.871,Z 628.348,A -85,B 0,C 180,E1 -14853.721,E2 -14853.721} C_VEL
LIN {X 0,Y 324.909,Z 625.853,A -85,B 0,C 180,E1 -14855.724,E2 -14855.724} C_VEL
LIN {X 0,Y 325.158,Z 622.778,A -85,B 0,C 180,E1 -14857.451,E2 -14857.451} C_VEL
LIN {X 0,Y 325.596,Z 618.434,A -85,B 0,C 180,E1 -14859.316,E2 -14859.316} C_VEL
LIN {X 0,Y 326.255,Z 612.903,A -85,B 0,C 180,E1 -14861.179,E2 -14861.179} C_VEL
LIN {X 0,Y 327.223,Z 606.002,A -85,B 0,C 180,E1 -14863.033,E2 -14863.033} C_VEL
LIN {X 0,Y 328.429,Z 597.366,A -85,B 0,C 180,E1 -14864.879,E2 -14864.879} C_VEL
LIN {X 0,Y 329.554,Z 588.708,A -85,B 0,C 180,E1 -14866.381,E2 -14866.381} C_VEL
LIN {X 0,Y 330.844,Z 578.792,A -85,B 0,C 180,E1 -14867.78,E2 -14867.78} C_VEL
LIN {X 0,Y 332.219,Z 568.16,A -85,B 0,C 180,E1 -14868.981,E2 -14868.981} C_VEL
LIN {X 0,Y 333.495,Z 556.271,A -85,B 0,C 180,E1 -14870.026,E2 -14870.026} C_VEL
LIN {X 0,Y 334.619,Z 543.898,A -85,B 0,C 180,E1 -14870.839,E2 -14870.839} C_VEL
LIN {X 0,Y 335.529,Z 531.171,A -85,B 0,C 180,E1 -14871.423,E2 -14871.423} C_VEL
LIN {X 0,Y 336.062,Z 517.759,A -85,B 0,C 180,E1 -14871.79,E2 -14871.79} C_VEL
LIN {X 0,Y 337.117,Z 454.145,A -85,B 0,C 180,E1 -14873.153,E2 -14873.153} C_VEL
LIN {X 0,Y 332.544,Z 426.993,A -85,B 0,C 180,E1 -14874.114,E2 -14874.114} C_VEL
LIN {X 0,Y 330.817,Z 417.807,A -85,B 0,C 180,E1 -14874.474,E2 -14874.474} C_VEL
LIN {X 0,Y 330.963,Z 414.141,A -85,B 0,C 180,E1 -14875.468,E2 -14875.468} C_VEL
LIN {X 0,Y 328.64,Z 402.09,A -85,B 0,C 180,E1 -14879.032,E2 -14879.032} C_VEL
LIN {X 0,Y 326.62,Z 393.3,A -85,B 0,C 180,E1 -14881.815,E2 -14881.815} C_VEL
LIN {X 0,Y 326.614,Z 393.3,A -85,B 0,C 180,E1 -14885.519,E2 -14885.519} C_VEL
LIN {X 0,Y 326.612,Z 393.301,A -85,B 0,C 180,E1 -14889.227,E2 -14889.227} C_VEL
LIN {X 0,Y 326.583,Z 393.307,A -85,B 0,C 180,E1 -14892.973,E2 -14892.973} C_VEL
LIN {X 0,Y 326.583,Z 393.306,A -85,B 0,C 180,E1 -14897.027,E2 -14897.027} C_VEL
LIN {X 0,Y 326.612,Z 393.302,A -85,B 0,C 180,E1 -14900.773,E2 -14900.773} C_VEL
LIN {X 0,Y 326.614,Z 393.3,A -85,B 0,C 180,E1 -14904.48,E2 -14904.48} C_VEL
LIN {X 0,Y 326.609,Z 393.298,A -85,B 0,C 180,E1 -14907.456,E2 -14907.456} C_VEL
LIN {X 0,Y 326.649,Z 393.296,A -85,B 0,C 180,E1 -14910.34,E2 -14910.34} C_VEL
LIN {X 0,Y 326.691,Z 393.293,A -85,B 0,C 180,E1 -14914.516,E2 -14914.516} C_VEL
LIN {X 0,Y 326.65,Z 393.299,A -85,B 0,C 180,E1 -14918.546,E2 -14918.546} C_VEL
LIN {X 0,Y 326.746,Z 393.281,A -85,B 0,C 180,E1 -14921.178,E2 -14921.178} C_VEL
LIN {X 0,Y 326.765,Z 393.277,A -85,B 0,C 180,E1 -14925.433,E2 -14925.433} C_VEL
LIN {X 0,Y 326.775,Z 393.278,A -85,B 0,C 180,E1 -14928.839,E2 -14928.839} C_VEL
LIN {X 0,Y 326.946,Z 393.26,A -85,B 0,C 180,E1 -14932.59,E2 -14932.59} C_VEL
LIN {X 0,Y 326.986,Z 393.253,A -85,B 0,C 180,E1 -14933.831,E2 -14933.831} C_VEL
LIN {X 0,Y 327.048,Z 393.244,A -85,B 0,C 180,E1 -14937.537,E2 -14937.537} C_VEL
LIN {X 0,Y 327.2,Z 393.228,A -85,B 0,C 180,E1 -14940,E2 -14940} C_VEL
LIN {X 0,Y 327.051,Z 393.246,A -85,B 0,C 180,E1 -14942.463,E2 -14942.463} C_VEL
LIN {X 0,Y 326.974,Z 393.252,A -85,B 0,C 180,E1 -14946.664,E2 -14946.664} C_VEL
LIN {X 0,Y 326.816,Z 393.277,A -85,B 0,C 180,E1 -14949.906,E2 -14949.906} C_VEL
LIN {X 0,Y 326.761,Z 393.281,A -85,B 0,C 180,E1 -14953.685,E2 -14953.685} C_VEL
LIN {X 0,Y 326.702,Z 393.286,A -85,B 0,C 180,E1 -14957.528,E2 -14957.528} C_VEL
LIN {X 0,Y 326.675,Z 393.293,A -85,B 0,C 180,E1 -14960.134,E2 -14960.134} C_VEL
LIN {X 0,Y 326.655,Z 393.295,A -85,B 0,C 180,E1 -14964.129,E2 -14964.129} C_VEL
LIN {X 0,Y 326.687,Z 393.288,A -85,B 0,C 180,E1 -14966.858,E2 -14966.858} C_VEL
LIN {X 0,Y 326.641,Z 393.293,A -85,B 0,C 180,E1 -14970.611,E2 -14970.611} C_VEL
LIN {X 0,Y 326.609,Z 393.3,A -85,B 0,C 180,E1 -14974.019,E2 -14974.019} C_VEL
LIN {X 0,Y 326.631,Z 393.297,A -85,B 0,C 180,E1 -14977.239,E2 -14977.239} C_VEL
LIN {X 0,Y 326.601,Z 393.299,A -85,B 0,C 180,E1 -14980.208,E2 -14980.208} C_VEL
LIN {X 0,Y 326.565,Z 393.308,A -85,B 0,C 180,E1 -14983.525,E2 -14983.525} C_VEL
LIN {X 0,Y 326.578,Z 393.304,A -85,B 0,C 180,E1 -14987.028,E2 -14987.028} C_VEL
LIN {X 0,Y 326.613,Z 393.299,A -85,B 0,C 180,E1 -14990.773,E2 -14990.773} C_VEL
LIN {X 0,Y 326.614,Z 393.298,A -85,B 0,C 180,E1 -14994.481,E2 -14994.481} C_VEL
LIN {X 0,Y 326.612,Z 393.302,A -85,B 0,C 180,E1 -14997.456,E2 -14997.456} C_VEL
LIN {X 0,Y 326.662,Z 393.293,A -85,B 0,C 180,E1 -15000.341,E2 -15000.341} C_VEL
LIN {X 0,Y 326.676,Z 393.312,A -85,B 0,C 180,E1 -15001.817,E2 -15001.817} C_VEL
LIN {X 0,Y 328.802,Z 403.362,A -85,B 0,C 180,E1 -15005.166,E2 -15005.166} C_VEL
LIN {X 0,Y 328.964,Z 404.259,A -85,B 0,C 180,E1 -15005.451,E2 -15005.451} C_VEL
LIN {X 0,Y 334.571,Z 419.204,A -85,B 0,C 180,E1 -15006.237,E2 -15006.237} C_VEL
LIN {X 0,Y 337.669,Z 435.311,A -85,B 0,C 180,E1 -15006.836,E2 -15006.836} C_VEL
LIN {X 0,Y 336.231,Z 502.85,A -85,B 0,C 180,E1 -15008.262,E2 -15008.262} C_VEL
LIN {X 0,Y 335.82,Z 516.34,A -85,B 0,C 180,E1 -15008.637,E2 -15008.637} C_VEL
LIN {X 0,Y 334.96,Z 529.733,A -85,B 0,C 180,E1 -15009.264,E2 -15009.264} C_VEL
LIN {X 0,Y 334.057,Z 540.946,A -85,B 0,C 180,E1 -15010.009,E2 -15010.009} C_VEL
LIN {X 0,Y 332.883,Z 552.935,A -85,B 0,C 180,E1 -15011.058,E2 -15011.058} C_VEL
LIN {X 0,Y 331.634,Z 563.609,A -85,B 0,C 180,E1 -15012.264,E2 -15012.264} C_VEL
LIN {X 0,Y 330.463,Z 573.707,A -85,B 0,C 180,E1 -15013.695,E2 -15013.695} C_VEL
LIN {X 0,Y 329.22,Z 582.171,A -85,B 0,C 180,E1 -15015.157,E2 -15015.157} C_VEL
LIN {X 0,Y 327.899,Z 590.798,A -85,B 0,C 180,E1 -15016.994,E2 -15016.994} C_VEL
LIN {X 0,Y 326.901,Z 597.674,A -85,B 0,C 180,E1 -15018.844,E2 -15018.844} C_VEL
LIN {X 0,Y 326.111,Z 603.178,A -85,B 0,C 180,E1 -15020.699,E2 -15020.699} C_VEL
LIN {X 0,Y 325.588,Z 607.498,A -85,B 0,C 180,E1 -15022.559,E2 -15022.559} C_VEL
LIN {X 0,Y 325.322,Z 609.783,A -85,B 0,C 180,E1 -15023.799,E2 -15023.799} C_VEL
LIN {X 0,Y 325.182,Z 611.641,A -85,B 0,C 180,E1 -15025.041,E2 -15025.041} C_VEL
LIN {X 0,Y 325.032,Z 613.039,A -85,B 0,C 180,E1 -15026.281,E2 -15026.281} C_VEL
LIN {X 0,Y 324.855,Z 614.647,A -85,B 0,C 180,E1 -15028.761,E2 -15028.761} C_VEL
LIN {X 0,Y 324.834,Z 614.879,A -85,B 0,C 180,E1 -15030,E2 -15030} C_VEL
LIN {X 0,Y 324.855,Z 614.688,A -85,B 0,C 180,E1 -15031.24,E2 -15031.24} C_VEL
LIN {X 0,Y 325.03,Z 613.132,A -85,B 0,C 180,E1 -15033.72,E2 -15033.72} C_VEL
LIN {X 0,Y 325.177,Z 611.774,A -85,B 0,C 180,E1 -15034.96,E2 -15034.96} C_VEL
LIN {X 0,Y 325.368,Z 609.487,A -85,B 0,C 180,E1 -15036.48,E2 -15036.48} C_VEL
LIN {X 0,Y 325.88,Z 605.014,A -85,B 0,C 180,E1 -15038.683,E2 -15038.683} C_VEL
LIN {X 0,Y 326.592,Z 599.992,A -85,B 0,C 180,E1 -15040.54,E2 -15040.54} C_VEL
LIN {X 0,Y 327.5,Z 593.669,A -85,B 0,C 180,E1 -15042.392,E2 -15042.392} C_VEL
LIN {X 0,Y 328.639,Z 585.755,A -85,B 0,C 180,E1 -15044.237,E2 -15044.237} C_VEL
LIN {X 0,Y 330.115,Z 575.909,A -85,B 0,C 180,E1 -15046.068,E2 -15046.068} C_VEL
LIN {X 0,Y 331.363,Z 565.575,A -85,B 0,C 180,E1 -15047.592,E2 -15047.592} C_VEL
LIN {X 0,Y 332.604,Z 555.337,A -85,B 0,C 180,E1 -15048.799,E2 -15048.799} C_VEL
LIN {X 0,Y 333.82,Z 544.131,A -85,B 0,C 180,E1 -15049.846,E2 -15049.846} C_VEL
LIN {X 0,Y 334.848,Z 532.753,A -85,B 0,C 180,E1 -15050.663,E2 -15050.663} C_VEL
LIN {X 0,Y 335.664,Z 519.743,A -85,B 0,C 180,E1 -15051.334,E2 -15051.334} C_VEL
LIN {X 0,Y 336.189,Z 507.287,A -85,B 0,C 180,E1 -15051.741,E2 -15051.741} C_VEL
LIN {X 0,Y 337.601,Z 434.379,A -85,B 0,C 180,E1 -15053.3,E2 -15053.3} C_VEL
LIN {X 0,Y 334.253,Z 417.966,A -85,B 0,C 180,E1 -15053.926,E2 -15053.926} C_VEL
LIN {X 0,Y 328.953,Z 404.183,A -85,B 0,C 180,E1 -15054.677,E2 -15054.677} C_VEL
LIN {X 0,Y 326.848,Z 394.103,A -85,B 0,C 180,E1 -15058.027,E2 -15058.027} C_VEL
LIN {X 0,Y 326.399,Z 393.404,A -85,B 0,C 180,E1 -15058.494,E2 -15058.494} C_VEL
LIN {X 0,Y 324.051,Z 393.62,A -85,B 0,C 180,E1 -15059.98,E2 -15059.98} C_VEL
LIN {X 0,Y 320.614,Z 394.201,A -85,B 0,C 180,E1 -15062.04,E2 -15062.04} C_VEL
LIN {X 0,Y 319.569,Z 394.176,A -85,B 0,C 180,E1 -15063.481,E2 -15063.481} C_VEL
LIN {X 0,Y 319.562,Z 394.177,A -85,B 0,C 180,E1 -15066.428,E2 -15066.428} C_VEL
LIN {X 0,Y 319.561,Z 394.177,A -85,B 0,C 180,E1 -15069.669,E2 -15069.669} C_VEL
LIN {X 0,Y 319.562,Z 394.176,A -85,B 0,C 180,E1 -15073.468,E2 -15073.468} C_VEL
LIN {X 0,Y 319.565,Z 394.178,A -85,B 0,C 180,E1 -15077.018,E2 -15077.018} C_VEL
LIN {X 0,Y 319.585,Z 394.171,A -85,B 0,C 180,E1 -15080.376,E2 -15080.376} C_VEL
LIN {X 0,Y 319.585,Z 394.178,A -85,B 0,C 180,E1 -15084.457,E2 -15084.457} C_VEL
LIN {X 0,Y 319.537,Z 394.183,A -85,B 0,C 180,E1 -15088.139,E2 -15088.139} C_VEL
LIN {X 0,Y 319.62,Z 394.168,A -85,B 0,C 180,E1 -15091.588,E2 -15091.588} C_VEL
LIN {X 0,Y 319.609,Z 394.167,A -85,B 0,C 180,E1 -15095.304,E2 -15095.304} C_VEL
LIN {X 0,Y 319.626,Z 394.168,A -85,B 0,C 180,E1 -15099.402,E2 -15099.402} C_VEL
LIN {X 0,Y 319.663,Z 394.166,A -85,B 0,C 180,E1 -15102.073,E2 -15102.073} C_VEL
LIN {X 0,Y 319.737,Z 394.156,A -85,B 0,C 180,E1 -15106.008,E2 -15106.008} C_VEL
LIN {X 0,Y 319.762,Z 394.156,A -85,B 0,C 180,E1 -15109.873,E2 -15109.873} C_VEL
LIN {X 0,Y 319.938,Z 394.127,A -85,B 0,C 180,E1 -15112.426,E2 -15112.426} C_VEL
LIN {X 0,Y 319.753,Z 394.152,A -85,B 0,C 180,E1 -15114.956,E2 -15114.956} C_VEL
LIN {X 0,Y 319.995,Z 394.124,A -85,B 0,C 180,E1 -15117.482,E2 -15117.482} C_VEL
LIN {X 0,Y 320.154,Z 394.105,A -85,B 0,C 180,E1 -15120,E2 -15120} C_VEL
LIN {X 0,Y 319.995,Z 394.123,A -85,B 0,C 180,E1 -15122.518,E2 -15122.518} C_VEL
LIN {X 0,Y 319.943,Z 394.128,A -85,B 0,C 180,E1 -15126.306,E2 -15126.306} C_VEL
LIN {X 0,Y 319.758,Z 394.152,A -85,B 0,C 180,E1 -15130.127,E2 -15130.127} C_VEL
LIN {X 0,Y 319.735,Z 394.155,A -85,B 0,C 180,E1 -15134.724,E2 -15134.724} C_VEL
LIN {X 0,Y 319.693,Z 394.161,A -85,B 0,C 180,E1 -15139.038,E2 -15139.038} C_VEL
LIN {X 0,Y 319.575,Z 394.176,A -85,B 0,C 180,E1 -15143.319,E2 -15143.319} C_VEL
LIN {X 0,Y 319.638,Z 394.167,A -85,B 0,C 180,E1 -15146.088,E2 -15146.088} C_VEL
LIN {X 0,Y 319.583,Z 394.175,A -85,B 0,C 180,E1 -15148.934,E2 -15148.934} C_VEL
LIN {X 0,Y 319.534,Z 394.18,A -85,B 0,C 180,E1 -15151.862,E2 -15151.862} C_VEL
LIN {X 0,Y 319.583,Z 394.176,A -85,B 0,C 180,E1 -15155.543,E2 -15155.543} C_VEL
LIN {X 0,Y 319.561,Z 394.177,A -85,B 0,C 180,E1 -15159.668,E2 -15159.668} C_VEL
LIN {X 0,Y 319.56,Z 394.179,A -85,B 0,C 180,E1 -15163.467,E2 -15163.467} C_VEL
LIN {X 0,Y 319.564,Z 394.181,A -85,B 0,C 180,E1 -15167.017,E2 -15167.017} C_VEL
LIN {X 0,Y 319.55,Z 394.179,A -85,B 0,C 180,E1 -15170.371,E2 -15170.371} C_VEL
LIN {X 0,Y 319.561,Z 394.179,A -85,B 0,C 180,E1 -15173.572,E2 -15173.572} C_VEL
LIN {X 0,Y 319.597,Z 394.283,A -85,B 0,C 180,E1 -15177.773,E2 -15177.773} C_VEL
LIN {X 0,Y 322.117,Z 405.43,A -85,B 0,C 180,E1 -15181.314,E2 -15181.314} C_VEL
LIN {X 0,Y 324.141,Z 416.507,A -85,B 0,C 180,E1 -15184.645,E2 -15184.645} C_VEL
LIN {X 0,Y 324.058,Z 417.628,A -85,B 0,C 180,E1 -15184.954,E2 -15184.954} C_VEL
LIN {X 0,Y 328.896,Z 443.852,A -85,B 0,C 180,E1 -15185.977,E2 -15185.977} C_VEL
LIN {X 0,Y 330.802,Z 456.323,A -85,B 0,C 180,E1 -15186.412,E2 -15186.412} C_VEL
LIN {X 0,Y 329.188,Z 525.922,A -85,B 0,C 180,E1 -15187.937,E2 -15187.937} C_VEL
LIN {X 0,Y 328.4,Z 539.111,A -85,B 0,C 180,E1 -15188.459,E2 -15188.459} C_VEL
LIN {X 0,Y 327.376,Z 551.228,A -85,B 0,C 180,E1 -15189.172,E2 -15189.172} C_VEL
LIN {X 0,Y 326.05,Z 563.458,A -85,B 0,C 180,E1 -15190.154,E2 -15190.154} C_VEL
LIN {X 0,Y 324.625,Z 575.034,A -85,B 0,C 180,E1 -15191.377,E2 -15191.377} C_VEL
LIN {X 0,Y 323.131,Z 585.779,A -85,B 0,C 180,E1 -15192.811,E2 -15192.811} C_VEL
LIN {X 0,Y 321.995,Z 594.296,A -85,B 0,C 180,E1 -15194.224,E2 -15194.224} C_VEL
LIN {X 0,Y 320.716,Z 603.226,A -85,B 0,C 180,E1 -15196.051,E2 -15196.051} C_VEL
LIN {X 0,Y 319.529,Z 610.651,A -85,B 0,C 180,E1 -15197.939,E2 -15197.939} C_VEL
LIN {X 0,Y 318.764,Z 616.618,A -85,B 0,C 180,E1 -15199.841,E2 -15199.841} C_VEL
LIN {X 0,Y 318.234,Z 621.334,A -85,B 0,C 180,E1 -15201.746,E2 -15201.746} C_VEL
LIN {X 0,Y 317.89,Z 624.938,A -85,B 0,C 180,E1 -15203.653,E2 -15203.653} C_VEL
LIN {X 0,Y 317.794,Z 626.797,A -85,B 0,C 180,E1 -15204.925,E2 -15204.925} C_VEL
LIN {X 0,Y 317.78,Z 628.192,A -85,B 0,C 180,E1 -15206.195,E2 -15206.195} C_VEL
LIN {X 0,Y 317.751,Z 629.188,A -85,B 0,C 180,E1 -15207.464,E2 -15207.464} C_VEL
LIN {X 0,Y 317.723,Z 629.794,A -85,B 0,C 180,E1 -15208.732,E2 -15208.732} C_VEL
LIN {X 0,Y 317.738,Z 630.008,A -85,B 0,C 180,E1 -15210,E2 -15210} C_VEL
LIN {X 0,Y 317.723,Z 629.788,A -85,B 0,C 180,E1 -15211.267,E2 -15211.267} C_VEL
LIN {X 0,Y 317.751,Z 629.179,A -85,B 0,C 180,E1 -15212.535,E2 -15212.535} C_VEL
LIN {X 0,Y 317.78,Z 628.18,A -85,B 0,C 180,E1 -15213.804,E2 -15213.804} C_VEL
LIN {X 0,Y 317.826,Z 625.918,A -85,B 0,C 180,E1 -15215.688,E2 -15215.688} C_VEL
LIN {X 0,Y 318.087,Z 622.609,A -85,B 0,C 180,E1 -15217.618,E2 -15217.618} C_VEL
LIN {X 0,Y 318.577,Z 618.266,A -85,B 0,C 180,E1 -15219.523,E2 -15219.523} C_VEL
LIN {X 0,Y 319.242,Z 612.733,A -85,B 0,C 180,E1 -15221.428,E2 -15221.428} C_VEL
LIN {X 0,Y 320.295,Z 605.833,A -85,B 0,C 180,E1 -15223.32,E2 -15223.32} C_VEL
LIN {X 0,Y 321.363,Z 598.786,A -85,B 0,C 180,E1 -15224.89,E2 -15224.89} C_VEL
LIN {X 0,Y 322.493,Z 590.117,A -85,B 0,C 180,E1 -15226.487,E2 -15226.487} C_VEL
LIN {X 0,Y 323.914,Z 579.797,A -85,B 0,C 180,E1 -15228.01,E2 -15228.01} C_VEL
LIN {X 0,Y 325.497,Z 567.988,A -85,B 0,C 180,E1 -15229.388,E2 -15229.388} C_VEL
LIN {X 0,Y 326.821,Z 556.097,A -85,B 0,C 180,E1 -15230.453,E2 -15230.453} C_VEL
LIN {X 0,Y 327.972,Z 543.723,A -85,B 0,C 180,E1 -15231.281,E2 -15231.281} C_VEL
LIN {X 0,Y 328.938,Z 530.993,A -85,B 0,C 180,E1 -15231.874,E2 -15231.874} C_VEL
LIN {X 0,Y 329.496,Z 517.572,A -85,B 0,C 180,E1 -15232.247,E2 -15232.247} C_VEL
LIN {X 0,Y 330.59,Z 454.957,A -85,B 0,C 180,E1 -15233.614,E2 -15233.614} C_VEL
LIN {X 0,Y 325.913,Z 427.366,A -85,B 0,C 180,E1 -15234.624,E2 -15234.624} C_VEL
LIN {X 0,Y 324.068,Z 417.604,A -85,B 0,C 180,E1 -15235.027,E2 -15235.027} C_VEL
LIN {X 0,Y 323.777,Z 414.063,A -85,B 0,C 180,E1 -15236.047,E2 -15236.047} C_VEL
LIN {X 0,Y 321.813,Z 403.918,A -85,B 0,C 180,E1 -15239.126,E2 -15239.126} C_VEL
LIN {X 0,Y 319.589,Z 394.176,A -85,B 0,C 180,E1 -15242.274,E2 -15242.274} C_VEL
LIN {X 0,Y 319.56,Z 394.178,A -85,B 0,C 180,E1 -15246.427,E2 -15246.427} C_VEL
LIN {X 0,Y 319.559,Z 394.178,A -85,B 0,C 180,E1 -15249.669,E2 -15249.669} C_VEL
LIN {X 0,Y 319.558,Z 394.177,A -85,B 0,C 180,E1 -15253.467,E2 -15253.467} C_VEL
LIN {X 0,Y 319.562,Z 394.18,A -85,B 0,C 180,E1 -15257.018,E2 -15257.018} C_VEL
LIN {X 0,Y 319.548,Z 394.179,A -85,B 0,C 180,E1 -15260.371,E2 -15260.371} C_VEL
LIN {X 0,Y 319.581,Z 394.176,A -85,B 0,C 180,E1 -15264.457,E2 -15264.457} C_VEL
LIN {X 0,Y 319.532,Z 394.181,A -85,B 0,C 180,E1 -15268.138,E2 -15268.138} C_VEL
LIN {X 0,Y 319.612,Z 394.169,A -85,B 0,C 180,E1 -15271.59,E2 -15271.59} C_VEL
LIN {X 0,Y 319.606,Z 394.17,A -85,B 0,C 180,E1 -15275.304,E2 -15275.304} C_VEL
LIN {X 0,Y 319.599,Z 394.173,A -85,B 0,C 180,E1 -15278.048,E2 -15278.048} C_VEL
LIN {X 0,Y 319.69,Z 394.161,A -85,B 0,C 180,E1 -15280.962,E2 -15280.962} C_VEL
LIN {X 0,Y 319.732,Z 394.153,A -85,B 0,C 180,E1 -15285.276,E2 -15285.276} C_VEL
LIN {X 0,Y 319.755,Z 394.153,A -85,B 0,C 180,E1 -15289.873,E2 -15289.873} C_VEL
LIN {X 0,Y 319.939,Z 394.13,A -85,B 0,C 180,E1 -15293.694,E2 -15293.694} C_VEL
LIN {X 0,Y 319.992,Z 394.122,A -85,B 0,C 180,E1 -15297.482,E2 -15297.482} C_VEL
LIN {X 0,Y 320.151,Z 394.106,A -85,B 0,C 180,E1 -15300,E2 -15300} C_VEL
LIN {X 0,Y 319.994,Z 394.125,A -85,B 0,C 180,E1 -15302.518,E2 -15302.518} C_VEL
LIN {X 0,Y 319.934,Z 394.129,A -85,B 0,C 180,E1 -15306.654,E2 -15306.654} C_VEL
LIN {X 0,Y 319.76,Z 394.155,A -85,B 0,C 180,E1 -15310.127,E2 -15310.127} C_VEL
LIN {X 0,Y 319.733,Z 394.155,A -85,B 0,C 180,E1 -15314.724,E2 -15314.724} C_VEL
LIN {X 0,Y 319.693,Z 394.16,A -85,B 0,C 180,E1 -15319.039,E2 -15319.039} C_VEL
LIN {X 0,Y 319.573,Z 394.176,A -85,B 0,C 180,E1 -15323.319,E2 -15323.319} C_VEL
LIN {X 0,Y 319.637,Z 394.169,A -85,B 0,C 180,E1 -15326.088,E2 -15326.088} C_VEL
LIN {X 0,Y 319.591,Z 394.173,A -85,B 0,C 180,E1 -15328.934,E2 -15328.934} C_VEL
LIN {X 0,Y 319.535,Z 394.184,A -85,B 0,C 180,E1 -15331.862,E2 -15331.862} C_VEL
LIN {X 0,Y 319.582,Z 394.177,A -85,B 0,C 180,E1 -15335.543,E2 -15335.543} C_VEL
LIN {X 0,Y 319.583,Z 394.178,A -85,B 0,C 180,E1 -15339.624,E2 -15339.624} C_VEL
LIN {X 0,Y 319.524,Z 394.185,A -85,B 0,C 180,E1 -15343.461,E2 -15343.461} C_VEL
LIN {X 0,Y 319.556,Z 394.178,A -85,B 0,C 180,E1 -15347.017,E2 -15347.017} C_VEL
LIN {X 0,Y 319.549,Z 394.179,A -85,B 0,C 180,E1 -15350.371,E2 -15350.371} C_VEL
LIN {X 0,Y 319.561,Z 394.18,A -85,B 0,C 180,E1 -15353.573,E2 -15353.573} C_VEL
LIN {X 0,Y 319.579,Z 394.176,A -85,B 0,C 180,E1 -15356.687,E2 -15356.687} C_VEL
LIN {X 0,Y 319.593,Z 394.172,A -85,B 0,C 180,E1 -15359.617,E2 -15359.617} C_VEL
LIN {X 0,Y 319.622,Z 394.259,A -85,B 0,C 180,E1 -15361.392,E2 -15361.392} C_VEL
LIN {X 0,Y 321.663,Z 403.751,A -85,B 0,C 180,E1 -15364.642,E2 -15364.642} C_VEL
LIN {X 0,Y 321.866,Z 404.629,A -85,B 0,C 180,E1 -15364.876,E2 -15364.876} C_VEL
LIN {X 0,Y 328.364,Z 421.708,A -85,B 0,C 180,E1 -15365.814,E2 -15365.814} C_VEL
LIN {X 0,Y 331.135,Z 436.517,A -85,B 0,C 180,E1 -15366.375,E2 -15366.375} C_VEL
LIN {X 0,Y 329.666,Z 503.041,A -85,B 0,C 180,E1 -15367.806,E2 -15367.806} C_VEL
LIN {X 0,Y 329.24,Z 516.52,A -85,B 0,C 180,E1 -15368.188,E2 -15368.188} C_VEL
LIN {X 0,Y 328.343,Z 529.909,A -85,B 0,C 180,E1 -15368.826,E2 -15368.826} C_VEL
LIN {X 0,Y 327.412,Z 541.12,A -85,B 0,C 180,E1 -15369.586,E2 -15369.586} C_VEL
LIN {X 0,Y 326.171,Z 553.108,A -85,B 0,C 180,E1 -15370.653,E2 -15370.653} C_VEL
LIN {X 0,Y 324.88,Z 563.78,A -85,B 0,C 180,E1 -15371.883,E2 -15371.883} C_VEL
LIN {X 0,Y 323.64,Z 574.044,A -85,B 0,C 180,E1 -15373.37,E2 -15373.37} C_VEL
LIN {X 0,Y 322.348,Z 582.341,A -85,B 0,C 180,E1 -15374.833,E2 -15374.833} C_VEL
LIN {X 0,Y 320.97,Z 590.968,A -85,B 0,C 180,E1 -15376.708,E2 -15376.708} C_VEL
LIN {X 0,Y 319.929,Z 597.843,A -85,B 0,C 180,E1 -15378.597,E2 -15378.597} C_VEL
LIN {X 0,Y 319.094,Z 603.347,A -85,B 0,C 180,E1 -15380.492,E2 -15380.492} C_VEL
LIN {X 0,Y 318.527,Z 607.666,A -85,B 0,C 180,E1 -15382.393,E2 -15382.393} C_VEL
LIN {X 0,Y 318.249,Z 609.951,A -85,B 0,C 180,E1 -15383.661,E2 -15383.661} C_VEL
LIN {X 0,Y 318.11,Z 611.808,A -85,B 0,C 180,E1 -15384.93,E2 -15384.93} C_VEL
LIN {X 0,Y 317.967,Z 613.207,A -85,B 0,C 180,E1 -15386.198,E2 -15386.198} C_VEL
LIN {X 0,Y 317.766,Z 614.814,A -85,B 0,C 180,E1 -15388.733,E2 -15388.733} C_VEL
LIN {X 0,Y 317.743,Z 615.046,A -85,B 0,C 180,E1 -15390,E2 -15390} C_VEL
LIN {X 0,Y 317.766,Z 614.854,A -85,B 0,C 180,E1 -15391.268,E2 -15391.268} C_VEL
LIN {X 0,Y 317.965,Z 613.298,A -85,B 0,C 180,E1 -15393.802,E2 -15393.802} C_VEL
LIN {X 0,Y 318.105,Z 611.94,A -85,B 0,C 180,E1 -15395.07,E2 -15395.07} C_VEL
LIN {X 0,Y 318.411,Z 609.072,A -85,B 0,C 180,E1 -15396.972,E2 -15396.972} C_VEL
LIN {X 0,Y 318.871,Z 605.18,A -85,B 0,C 180,E1 -15398.875,E2 -15398.875} C_VEL
LIN {X 0,Y 319.602,Z 600.158,A -85,B 0,C 180,E1 -15400.773,E2 -15400.773} C_VEL
LIN {X 0,Y 320.541,Z 593.835,A -85,B 0,C 180,E1 -15402.666,E2 -15402.666} C_VEL
LIN {X 0,Y 321.766,Z 585.92,A -85,B 0,C 180,E1 -15404.548,E2 -15404.548} C_VEL
LIN {X 0,Y 323.294,Z 576.073,A -85,B 0,C 180,E1 -15406.416,E2 -15406.416} C_VEL
LIN {X 0,Y 324.605,Z 565.738,A -85,B 0,C 180,E1 -15407.971,E2 -15407.971} C_VEL
LIN {X 0,Y 326.051,Z 554.077,A -85,B 0,C 180,E1 -15409.355,E2 -15409.355} C_VEL
LIN {X 0,Y 327.33,Z 542.452,A -85,B 0,C 180,E1 -15410.42,E2 -15410.42} C_VEL
LIN {X 0,Y 328.411,Z 530.356,A -85,B 0,C 180,E1 -15411.252,E2 -15411.252} C_VEL
LIN {X 0,Y 329.222,Z 517.153,A -85,B 0,C 180,E1 -15411.896,E2 -15411.896} C_VEL
LIN {X 0,Y 329.751,Z 504.238,A -85,B 0,C 180,E1 -15412.27,E2 -15412.27} C_VEL
LIN {X 0,Y 331.072,Z 435.387,A -85,B 0,C 180,E1 -15413.767,E2 -15413.767} C_VEL
LIN {X 0,Y 328.042,Z 420.457,A -85,B 0,C 180,E1 -15414.353,E2 -15414.353} C_VEL
LIN {X 0,Y 321.792,Z 404.352,A -85,B 0,C 180,E1 -15415.267,E2 -15415.267} C_VEL
LIN {X 0,Y 319.641,Z 394.17,A -85,B 0,C 180,E1 -15418.769,E2 -15418.769} C_VEL
LIN {X 0,Y 319.535,Z 394.182,A -85,B 0,C 180,E1 -15421.862,E2 -15421.862} C_VEL
LIN {X 0,Y 319.569,Z 394.176,A -85,B 0,C 180,E1 -15423.481,E2 -15423.481} C_VEL
LIN {X 0,Y 318.865,Z 394.268,A -85,B 0,C 180,E1 -15424.532,E2 -15424.532} C_VEL
LIN {X 0,Y 316.029,Z 394.62,A -85,B 0,C 180,E1 -15426.245,E2 -15426.245} C_VEL
LIN {X 0,Y 313.64,Z 394.921,A -85,B 0,C 180,E1 -15427.632,E2 -15427.632} C_VEL
LIN {X 0,Y 312.599,Z 395.049,A -85,B 0,C 180,E1 -15428.706,E2 -15428.706} C_VEL
LIN {X 0,Y 312.504,Z 395.058,A -85,B 0,C 180,E1 -15429.069,E2 -15429.069} C_VEL
LIN {X 0,Y 312.497,Z 395.061,A -85,B 0,C 180,E1 -15432.431,E2 -15432.431} C_VEL
LIN {X 0,Y 312.484,Z 395.059,A -85,B 0,C 180,E1 -15436.031,E2 -15436.031} C_VEL
LIN {X 0,Y 312.509,Z 395.052,A -85,B 0,C 180,E1 -15439.874,E2 -15439.874} C_VEL
LIN {X 0,Y 312.542,Z 395.054,A -85,B 0,C 180,E1 -15442.617,E2 -15442.617} C_VEL
LIN {X 0,Y 312.523,Z 395.055,A -85,B 0,C 180,E1 -15446.311,E2 -15446.311} C_VEL
LIN {X 0,Y 312.549,Z 395.052,A -85,B 0,C 180,E1 -15450.35,E2 -15450.35} C_VEL
LIN {X 0,Y 312.607,Z 395.046,A -85,B 0,C 180,E1 -15454.064,E2 -15454.064} C_VEL
LIN {X 0,Y 312.592,Z 395.045,A -85,B 0,C 180,E1 -15457.529,E2 -15457.529} C_VEL
LIN {X 0,Y 312.644,Z 395.037,A -85,B 0,C 180,E1 -15461.657,E2 -15461.657} C_VEL
LIN {X 0,Y 312.698,Z 395.032,A -85,B 0,C 180,E1 -15465.686,E2 -15465.686} C_VEL
LIN {X 0,Y 312.707,Z 395.033,A -85,B 0,C 180,E1 -15469.642,E2 -15469.642} C_VEL
LIN {X 0,Y 312.877,Z 395.007,A -85,B 0,C 180,E1 -15472.254,E2 -15472.254} C_VEL
LIN {X 0,Y 312.723,Z 395.028,A -85,B 0,C 180,E1 -15474.842,E2 -15474.842} C_VEL
LIN {X 0,Y 312.993,Z 394.991,A -85,B 0,C 180,E1 -15478.713,E2 -15478.713} C_VEL
LIN {X 0,Y 312.993,Z 394.995,A -85,B 0,C 180,E1 -15481.287,E2 -15481.287} C_VEL
LIN {X 0,Y 312.719,Z 395.027,A -85,B 0,C 180,E1 -15485.158,E2 -15485.158} C_VEL
LIN {X 0,Y 312.899,Z 395.005,A -85,B 0,C 180,E1 -15486.448,E2 -15486.448} C_VEL
LIN {X 0,Y 312.704,Z 395.029,A -85,B 0,C 180,E1 -15490.358,E2 -15490.358} C_VEL
LIN {X 0,Y 312.704,Z 395.031,A -85,B 0,C 180,E1 -15494.888,E2 -15494.888} C_VEL
LIN {X 0,Y 312.634,Z 395.041,A -85,B 0,C 180,E1 -15499.236,E2 -15499.236} C_VEL
LIN {X 0,Y 312.55,Z 395.047,A -85,B 0,C 180,E1 -15502.789,E2 -15502.789} C_VEL
LIN {X 0,Y 312.606,Z 395.044,A -85,B 0,C 180,E1 -15505.935,E2 -15505.935} C_VEL
LIN {X 0,Y 312.542,Z 395.053,A -85,B 0,C 180,E1 -15509.65,E2 -15509.65} C_VEL
LIN {X 0,Y 312.522,Z 395.055,A -85,B 0,C 180,E1 -15513.689,E2 -15513.689} C_VEL
LIN {X 0,Y 312.523,Z 395.056,A -85,B 0,C 180,E1 -15517.386,E2 -15517.386} C_VEL
LIN {X 0,Y 312.493,Z 395.058,A -85,B 0,C 180,E1 -15520.709,E2 -15520.709} C_VEL
LIN {X 0,Y 312.476,Z 395.06,A -85,B 0,C 180,E1 -15524.205,E2 -15524.205} C_VEL
LIN {X 0,Y 312.489,Z 395.059,A -85,B 0,C 180,E1 -15527.918,E2 -15527.918} C_VEL
LIN {X 0,Y 312.508,Z 395.056,A -85,B 0,C 180,E1 -15531.917,E2 -15531.917} C_VEL
LIN {X 0,Y 312.535,Z 395.054,A -85,B 0,C 180,E1 -15534.22,E2 -15534.22} C_VEL
LIN {X 0,Y 312.547,Z 395.076,A -85,B 0,C 180,E1 -15537.253,E2 -15537.253} C_VEL
LIN {X 0,Y 315.092,Z 406.485,A -85,B 0,C 180,E1 -15540.979,E2 -15540.979} C_VEL
LIN {X 0,Y 317.189,Z 417.541,A -85,B 0,C 180,E1 -15544.393,E2 -15544.393} C_VEL
LIN {X 0,Y 321.328,Z 438.396,A -85,B 0,C 180,E1 -15545.247,E2 -15545.247} C_VEL
LIN {X 0,Y 324.211,Z 456.602,A -85,B 0,C 180,E1 -15545.913,E2 -15545.913} C_VEL
LIN {X 0,Y 322.627,Z 525.768,A -85,B 0,C 180,E1 -15547.464,E2 -15547.464} C_VEL
LIN {X 0,Y 321.816,Z 538.953,A -85,B 0,C 180,E1 -15547.996,E2 -15547.996} C_VEL
LIN {X 0,Y 320.766,Z 551.068,A -85,B 0,C 180,E1 -15548.722,E2 -15548.722} C_VEL
LIN {X 0,Y 319.37,Z 563.295,A -85,B 0,C 180,E1 -15549.721,E2 -15549.721} C_VEL
LIN {X 0,Y 317.876,Z 574.87,A -85,B 0,C 180,E1 -15550.967,E2 -15550.967} C_VEL
LIN {X 0,Y 316.343,Z 585.292,A -85,B 0,C 180,E1 -15552.38,E2 -15552.38} C_VEL
LIN {X 0,Y 315.1,Z 594.477,A -85,B 0,C 180,E1 -15553.937,E2 -15553.937} C_VEL
LIN {X 0,Y 313.82,Z 603.061,A -85,B 0,C 180,E1 -15555.738,E2 -15555.738} C_VEL
LIN {X 0,Y 312.574,Z 610.485,A -85,B 0,C 180,E1 -15557.666,E2 -15557.666} C_VEL
LIN {X 0,Y 311.732,Z 616.451,A -85,B 0,C 180,E1 -15559.609,E2 -15559.609} C_VEL
LIN {X 0,Y 311.196,Z 621.168,A -85,B 0,C 180,E1 -15561.558,E2 -15561.558} C_VEL
LIN {X 0,Y 310.822,Z 624.771,A -85,B 0,C 180,E1 -15563.508,E2 -15563.508} C_VEL
LIN {X 0,Y 310.699,Z 626.63,A -85,B 0,C 180,E1 -15564.809,E2 -15564.809} C_VEL
LIN {X 0,Y 310.693,Z 628.026,A -85,B 0,C 180,E1 -15566.109,E2 -15566.109} C_VEL
LIN {X 0,Y 310.674,Z 629.021,A -85,B 0,C 180,E1 -15567.407,E2 -15567.407} C_VEL
LIN {X 0,Y 310.638,Z 629.628,A -85,B 0,C 180,E1 -15568.703,E2 -15568.703} C_VEL
LIN {X 0,Y 310.65,Z 629.841,A -85,B 0,C 180,E1 -15570,E2 -15570} C_VEL
LIN {X 0,Y 310.638,Z 629.621,A -85,B 0,C 180,E1 -15571.296,E2 -15571.296} C_VEL
LIN {X 0,Y 310.674,Z 629.011,A -85,B 0,C 180,E1 -15572.593,E2 -15572.593} C_VEL
LIN {X 0,Y 310.693,Z 628.013,A -85,B 0,C 180,E1 -15573.891,E2 -15573.891} C_VEL
LIN {X 0,Y 310.724,Z 626.03,A -85,B 0,C 180,E1 -15575.615,E2 -15575.615} C_VEL
LIN {X 0,Y 311.029,Z 622.44,A -85,B 0,C 180,E1 -15577.792,E2 -15577.792} C_VEL
LIN {X 0,Y 311.531,Z 618.096,A -85,B 0,C 180,E1 -15579.741,E2 -15579.741} C_VEL
LIN {X 0,Y 312.234,Z 612.563,A -85,B 0,C 180,E1 -15581.688,E2 -15581.688} C_VEL
LIN {X 0,Y 313.355,Z 605.663,A -85,B 0,C 180,E1 -15583.621,E2 -15583.621} C_VEL
LIN {X 0,Y 314.452,Z 598.616,A -85,B 0,C 180,E1 -15585.225,E2 -15585.225} C_VEL
LIN {X 0,Y 315.635,Z 590.12,A -85,B 0,C 180,E1 -15586.826,E2 -15586.826} C_VEL
LIN {X 0,Y 317.149,Z 579.626,A -85,B 0,C 180,E1 -15588.408,E2 -15588.408} C_VEL
LIN {X 0,Y 318.803,Z 567.817,A -85,B 0,C 180,E1 -15589.812,E2 -15589.812} C_VEL
LIN {X 0,Y 320.173,Z 555.924,A -85,B 0,C 180,E1 -15590.897,E2 -15590.897} C_VEL
LIN {X 0,Y 321.37,Z 543.548,A -85,B 0,C 180,E1 -15591.74,E2 -15591.74} C_VEL
LIN {X 0,Y 322.363,Z 530.815,A -85,B 0,C 180,E1 -15592.344,E2 -15592.344} C_VEL
LIN {X 0,Y 322.944,Z 517.384,A -85,B 0,C 180,E1 -15592.723,E2 -15592.723} C_VEL
LIN {X 0,Y 324.07,Z 455.947,A -85,B 0,C 180,E1 -15594.091,E2 -15594.091} C_VEL
LIN {X 0,Y 319.627,Z 429.304,A -85,B 0,C 180,E1 -15595.09,E2 -15595.09} C_VEL
LIN {X 0,Y 317.169,Z 417.442,A -85,B 0,C 180,E1 -15595.605,E2 -15595.605} C_VEL
LIN {X 0,Y 315.114,Z 406.403,A -85,B 0,C 180,E1 -15599.018,E2 -15599.018} C_VEL
LIN {X 0,Y 312.546,Z 395.054,A -85,B 0,C 180,E1 -15602.747,E2 -15602.747} C_VEL
LIN {X 0,Y 312.537,Z 395.052,A -85,B 0,C 180,E1 -15605.95,E2 -15605.95} C_VEL
LIN {X 0,Y 312.505,Z 395.056,A -85,B 0,C 180,E1 -15610.125,E2 -15610.125} C_VEL
LIN {X 0,Y 312.482,Z 395.057,A -85,B 0,C 180,E1 -15613.969,E2 -15613.969} C_VEL
LIN {X 0,Y 312.487,Z 395.057,A -85,B 0,C 180,E1 -15617.918,E2 -15617.918} C_VEL
LIN {X 0,Y 312.5,Z 395.059,A -85,B 0,C 180,E1 -15620.971,E2 -15620.971} C_VEL
LIN {X 0,Y 312.533,Z 395.053,A -85,B 0,C 180,E1 -15624.22,E2 -15624.22} C_VEL
LIN {X 0,Y 312.505,Z 395.056,A -85,B 0,C 180,E1 -15627.334,E2 -15627.334} C_VEL
LIN {X 0,Y 312.545,Z 395.051,A -85,B 0,C 180,E1 -15631.279,E2 -15631.279} C_VEL
LIN {X 0,Y 312.587,Z 395.049,A -85,B 0,C 180,E1 -15634.711,E2 -15634.711} C_VEL
LIN {X 0,Y 312.589,Z 395.045,A -85,B 0,C 180,E1 -15637.529,E2 -15637.529} C_VEL
LIN {X 0,Y 312.64,Z 395.038,A -85,B 0,C 180,E1 -15641.656,E2 -15641.656} C_VEL
LIN {X 0,Y 312.696,Z 395.029,A -85,B 0,C 180,E1 -15645.686,E2 -15645.686} C_VEL
LIN {X 0,Y 312.701,Z 395.03,A -85,B 0,C 180,E1 -15649.642,E2 -15649.642} C_VEL
LIN {X 0,Y 312.895,Z 395.007,A -85,B 0,C 180,E1 -15653.552,E2 -15653.552} C_VEL
LIN {X 0,Y 312.939,Z 395.001,A -85,B 0,C 180,E1 -15657.426,E2 -15657.426} C_VEL
LIN {X 0,Y 313.104,Z 394.984,A -85,B 0,C 180,E1 -15660,E2 -15660} C_VEL
LIN {X 0,Y 312.941,Z 395.003,A -85,B 0,C 180,E1 -15662.574,E2 -15662.574} C_VEL
LIN {X 0,Y 312.897,Z 395.006,A -85,B 0,C 180,E1 -15666.637,E2 -15666.637} C_VEL
LIN {X 0,Y 312.789,Z 395.02,A -85,B 0,C 180,E1 -15669.049,E2 -15669.049} C_VEL
LIN {X 0,Y 312.636,Z 395.038,A -85,B 0,C 180,E1 -15672.991,E2 -15672.991} C_VEL
LIN {X 0,Y 312.64,Z 395.041,A -85,B 0,C 180,E1 -15675.65,E2 -15675.65} C_VEL
LIN {X 0,Y 312.609,Z 395.046,A -85,B 0,C 180,E1 -15679.708,E2 -15679.708} C_VEL
LIN {X 0,Y 312.548,Z 395.049,A -85,B 0,C 180,E1 -15682.79,E2 -15682.79} C_VEL
LIN {X 0,Y 312.605,Z 395.045,A -85,B 0,C 180,E1 -15685.936,E2 -15685.936} C_VEL
LIN {X 0,Y 312.547,Z 395.054,A -85,B 0,C 180,E1 -15689.65,E2 -15689.65} C_VEL
LIN {X 0,Y 312.521,Z 395.056,A -85,B 0,C 180,E1 -15693.689,E2 -15693.689} C_VEL
LIN {X 0,Y 312.54,Z 395.054,A -85,B 0,C 180,E1 -15697.383,E2 -15697.383} C_VEL
LIN {X 0,Y 312.494,Z 395.056,A -85,B 0,C 180,E1 -15700.709,E2 -15700.709} C_VEL
LIN {X 0,Y 312.453,Z 395.062,A -85,B 0,C 180,E1 -15704.21,E2 -15704.21} C_VEL
LIN {X 0,Y 312.486,Z 395.06,A -85,B 0,C 180,E1 -15707.919,E2 -15707.919} C_VEL
LIN {X 0,Y 312.507,Z 395.057,A -85,B 0,C 180,E1 -15711.917,E2 -15711.917} C_VEL
LIN {X 0,Y 312.534,Z 395.053,A -85,B 0,C 180,E1 -15714.221,E2 -15714.221} C_VEL
LIN {X 0,Y 312.507,Z 395.059,A -85,B 0,C 180,E1 -15717.334,E2 -15717.334} C_VEL
LIN {X 0,Y 312.582,Z 395.231,A -85,B 0,C 180,E1 -15720.956,E2 -15720.956} C_VEL
LIN {X 0,Y 314.633,Z 404.568,A -85,B 0,C 180,E1 -15724.239,E2 -15724.239} C_VEL
LIN {X 0,Y 322.131,Z 423.889,A -85,B 0,C 180,E1 -15725.363,E2 -15725.363} C_VEL
LIN {X 0,Y 324.648,Z 437.023,A -85,B 0,C 180,E1 -15725.881,E2 -15725.881} C_VEL
LIN {X 0,Y 323.12,Z 503.232,A -85,B 0,C 180,E1 -15727.332,E2 -15727.332} C_VEL
LIN {X 0,Y 322.682,Z 516.7,A -85,B 0,C 180,E1 -15727.722,E2 -15727.722} C_VEL
LIN {X 0,Y 321.727,Z 530.085,A -85,B 0,C 180,E1 -15728.369,E2 -15728.369} C_VEL
LIN {X 0,Y 320.777,Z 541.293,A -85,B 0,C 180,E1 -15729.144,E2 -15729.144} C_VEL
LIN {X 0,Y 319.491,Z 553.28,A -85,B 0,C 180,E1 -15730.232,E2 -15730.232} C_VEL
LIN {X 0,Y 318.139,Z 563.951,A -85,B 0,C 180,E1 -15731.485,E2 -15731.485} C_VEL
LIN {X 0,Y 316.967,Z 573.15,A -85,B 0,C 180,E1 -15732.827,E2 -15732.827} C_VEL
LIN {X 0,Y 315.493,Z 582.511,A -85,B 0,C 180,E1 -15734.496,E2 -15734.496} C_VEL
LIN {X 0,Y 314.058,Z 591.137,A -85,B 0,C 180,E1 -15736.41,E2 -15736.41} C_VEL
LIN {X 0,Y 312.953,Z 598.012,A -85,B 0,C 180,E1 -15738.34,E2 -15738.34} C_VEL
LIN {X 0,Y 312.097,Z 603.516,A -85,B 0,C 180,E1 -15740.277,E2 -15740.277} C_VEL
LIN {X 0,Y 311.497,Z 607.834,A -85,B 0,C 180,E1 -15742.22,E2 -15742.22} C_VEL
LIN {X 0,Y 311.18,Z 610.238,A -85,B 0,C 180,E1 -15743.589,E2 -15743.589} C_VEL
LIN {X 0,Y 311.041,Z 611.976,A -85,B 0,C 180,E1 -15744.815,E2 -15744.815} C_VEL
LIN {X 0,Y 310.903,Z 613.374,A -85,B 0,C 180,E1 -15746.112,E2 -15746.112} C_VEL
LIN {X 0,Y 310.681,Z 614.981,A -85,B 0,C 180,E1 -15748.704,E2 -15748.704} C_VEL
LIN {X 0,Y 310.656,Z 615.213,A -85,B 0,C 180,E1 -15750,E2 -15750} C_VEL
LIN {X 0,Y 310.681,Z 615.021,A -85,B 0,C 180,E1 -15751.296,E2 -15751.296} C_VEL
LIN {X 0,Y 310.901,Z 613.465,A -85,B 0,C 180,E1 -15753.889,E2 -15753.889} C_VEL
